LIN {X 0,Y 672.579,Z 201.622,A -85,B 0,C 180,E1 -3473.113,E2 -3473.113} C_VEL
LIN {X 0,Y 679.346,Z 218.804,A -85,B 0,C 180,E1 -3474.693,E2 -3474.693} C_VEL
LIN {X 0,Y 682.037,Z 226.59,A -85,B 0,C 180,E1 -3475.434,E2 -3475.434} C_VEL
LIN {X 0,Y 680.752,Z 266.781,A -85,B 0,C 180,E1 -3478.375,E2 -3478.375} C_VEL
LIN {X 0,Y 679.52,Z 306.415,A -85,B 0,C 180,E1 -3481.238,E2 -3481.238} C_VEL
LIN {X 0,Y 679.485,Z 310.379,A -85,B 0,C 180,E1 -3481.504,E2 -3481.504} C_VEL
LIN {X 0,Y 681.228,Z 320.364,A -85,B 0,C 180,E1 -3481.706,E2 -3481.706} C_VEL
LIN {X 0,Y 679.45,Z 568.033,A -85,B 0,C 180,E1 -3484.516,E2 -3484.516} C_VEL
LIN {X 0,Y 679.106,Z 608.658,A -85,B 0,C 180,E1 -3485,E2 -3485} C_VEL
LIN {X 0,Y 678.694,Z 631.405,A -85,B 0,C 180,E1 -3485.414,E2 -3485.414} C_VEL
LIN {X 0,Y 678.15,Z 652.378,A -85,B 0,C 180,E1 -3485.964,E2 -3485.964} C_VEL
LIN {X 0,Y 677.64,Z 669.474,A -85,B 0,C 180,E1 -3486.522,E2 -3486.522} C_VEL
LIN {X 0,Y 677.053,Z 686.549,A -85,B 0,C 180,E1 -3487.19,E2 -3487.19} C_VEL
LIN {X 0,Y 676.5,Z 702.61,A -85,B 0,C 180,E1 -3487.931,E2 -3487.931} C_VEL
LIN {X 0,Y 675.912,Z 718.028,A -85,B 0,C 180,E1 -3488.75,E2 -3488.75} C_VEL
LIN {X 0,Y 675.272,Z 734.049,A -85,B 0,C 180,E1 -3489.727,E2 -3489.727} C_VEL
LIN {X 0,Y 674.601,Z 751.677,A -85,B 0,C 180,E1 -3490.969,E2 -3490.969} C_VEL
LIN {X 0,Y 673.925,Z 768.647,A -85,B 0,C 180,E1 -3492.382,E2 -3492.382} C_VEL
LIN {X 0,Y 673.437,Z 781.527,A -85,B 0,C 180,E1 -3493.614,E2 -3493.614} C_VEL
LIN {X 0,Y 673.036,Z 793.645,A -85,B 0,C 180,E1 -3494.931,E2 -3494.931} C_VEL
LIN {X 0,Y 672.65,Z 806.255,A -85,B 0,C 180,E1 -3496.504,E2 -3496.504} C_VEL
LIN {X 0,Y 672.335,Z 818.497,A -85,B 0,C 180,E1 -3498.331,E2 -3498.331} C_VEL
LIN {X 0,Y 672.156,Z 827.245,A -85,B 0,C 180,E1 -3499.89,E2 -3499.89} C_VEL
LIN {X 0,Y 672.032,Z 834.911,A -85,B 0,C 180,E1 -3501.53,E2 -3501.53} C_VEL
LIN {X 0,Y 671.95,Z 841.394,A -85,B 0,C 180,E1 -3503.249,E2 -3503.249} C_VEL
LIN {X 0,Y 671.913,Z 846.943,A -85,B 0,C 180,E1 -3505.22,E2 -3505.22} C_VEL
LIN {X 0,Y 671.901,Z 850.246,A -85,B 0,C 180,E1 -3507.014,E2 -3507.014} C_VEL
LIN {X 0,Y 671.897,Z 851.95,A -85,B 0,C 180,E1 -3508.636,E2 -3508.636} C_VEL
LIN {X 0,Y 671.9,Z 852.431,A -85,B 0,C 180,E1 -3510.426,E2 -3510.426} C_VEL
LIN {X 0,Y 671.909,Z 851.064,A -85,B 0,C 180,E1 -3512.473,E2 -3512.473} C_VEL
LIN {X 0,Y 671.923,Z 848.206,A -85,B 0,C 180,E1 -3514.267,E2 -3514.267} C_VEL
LIN {X 0,Y 671.94,Z 844.025,A -85,B 0,C 180,E1 -3515.979,E2 -3515.979} C_VEL
LIN {X 0,Y 671.981,Z 838.375,A -85,B 0,C 180,E1 -3517.696,E2 -3517.696} C_VEL
LIN {X 0,Y 672.106,Z 829.893,A -85,B 0,C 180,E1 -3519.678,E2 -3519.678} C_VEL
LIN {X 0,Y 672.271,Z 821.072,A -85,B 0,C 180,E1 -3521.322,E2 -3521.322} C_VEL
LIN {X 0,Y 672.494,Z 811.756,A -85,B 0,C 180,E1 -3522.799,E2 -3522.799} C_VEL
LIN {X 0,Y 672.852,Z 799.566,A -85,B 0,C 180,E1 -3524.457,E2 -3524.457} C_VEL
LIN {X 0,Y 673.329,Z 784.965,A -85,B 0,C 180,E1 -3526.123,E2 -3526.123} C_VEL
LIN {X 0,Y 673.81,Z 771.549,A -85,B 0,C 180,E1 -3527.443,E2 -3527.443} C_VEL
LIN {X 0,Y 674.343,Z 757.55,A -85,B 0,C 180,E1 -3528.65,E2 -3528.65} C_VEL
LIN {X 0,Y 674.979,Z 741.859,A -85,B 0,C 180,E1 -3529.835,E2 -3529.835} C_VEL
LIN {X 0,Y 675.763,Z 721.934,A -85,B 0,C 180,E1 -3531.118,E2 -3531.118} C_VEL
LIN {X 0,Y 676.425,Z 704.738,A -85,B 0,C 180,E1 -3532.053,E2 -3532.053} C_VEL
LIN {X 0,Y 676.991,Z 688.587,A -85,B 0,C 180,E1 -3532.812,E2 -3532.812} C_VEL
LIN {X 0,Y 677.555,Z 671.856,A -85,B 0,C 180,E1 -3533.481,E2 -3533.481} C_VEL
LIN {X 0,Y 678.053,Z 655.221,A -85,B 0,C 180,E1 -3534.04,E2 -3534.04} C_VEL
LIN {X 0,Y 678.51,Z 638.285,A -85,B 0,C 180,E1 -3534.506,E2 -3534.506} C_VEL
LIN {X 0,Y 678.88,Z 621.075,A -85,B 0,C 180,E1 -3534.88,E2 -3534.88} C_VEL
LIN {X 0,Y 679.16,Z 603.568,A -85,B 0,C 180,E1 -3535.16,E2 -3535.16} C_VEL
LIN {X 0,Y 681.182,Z 326.681,A -85,B 0,C 180,E1 -3538.313,E2 -3538.313} C_VEL
LIN {X 0,Y 681.006,Z 317.975,A -85,B 0,C 180,E1 -3538.425,E2 -3538.425} C_VEL
LIN {X 0,Y 679.405,Z 309.493,A -85,B 0,C 180,E1 -3538.623,E2 -3538.623} C_VEL
LIN {X 0,Y 680.471,Z 276.701,A -85,B 0,C 180,E1 -3540.999,E2 -3540.999} C_VEL
LIN {X 0,Y 681.79,Z 234.937,A -85,B 0,C 180,E1 -3544.043,E2 -3544.043} C_VEL
LIN {X 0,Y 681.872,Z 225.908,A -85,B 0,C 180,E1 -3544.716,E2 -3544.716} C_VEL
LIN {X 0,Y 675.939,Z 210.334,A -85,B 0,C 180,E1 -3546.202,E2 -3546.202} C_VEL
LIN {X 0,Y 672.552,Z 201.457,A -85,B 0,C 180,E1 -3547.022,E2 -3547.022} C_VEL
LIN {X 0,Y 672.581,Z 201.453,A -85,B 0,C 180,E1 -3549.958,E2 -3549.958} C_VEL
LIN {X 0,Y 672.558,Z 201.452,A -85,B 0,C 180,E1 -3552.915,E2 -3552.915} C_VEL
LIN {X 0,Y 672.581,Z 201.448,A -85,B 0,C 180,E1 -3555.913,E2 -3555.913} C_VEL
LIN {X 0,Y 672.561,Z 201.45,A -85,B 0,C 180,E1 -3558.919,E2 -3558.919} C_VEL
LIN {X 0,Y 672.58,Z 201.45,A -85,B 0,C 180,E1 -3561.905,E2 -3561.905} C_VEL
LIN {X 0,Y 672.565,Z 201.448,A -85,B 0,C 180,E1 -3564.98,E2 -3564.98} C_VEL
LIN {X 0,Y 672.578,Z 201.451,A -85,B 0,C 180,E1 -3567.945,E2 -3567.945} C_VEL
LIN {X 0,Y 672.57,Z 201.443,A -85,B 0,C 180,E1 -3570.946,E2 -3570.946} C_VEL
LIN {X 0,Y 672.575,Z 201.452,A -85,B 0,C 180,E1 -3573.987,E2 -3573.987} C_VEL
LIN {X 0,Y 672.573,Z 201.435,A -85,B 0,C 180,E1 -3576.984,E2 -3576.984} C_VEL
LIN {X 0,Y 672.572,Z 201.448,A -85,B 0,C 180,E1 -3580.005,E2 -3580.005} C_VEL
LIN {X 0,Y 672.574,Z 201.438,A -85,B 0,C 180,E1 -3583.059,E2 -3583.059} C_VEL
LIN {X 0,Y 672.569,Z 201.445,A -85,B 0,C 180,E1 -3586.064,E2 -3586.064} C_VEL
LIN {X 0,Y 672.576,Z 201.439,A -85,B 0,C 180,E1 -3589.117,E2 -3589.117} C_VEL
LIN {X 0,Y 672.565,Z 201.446,A -85,B 0,C 180,E1 -3592.139,E2 -3592.139} C_VEL
LIN {X 0,Y 672.579,Z 201.437,A -85,B 0,C 180,E1 -3595.139,E2 -3595.139} C_VEL
LIN {X 0,Y 672.561,Z 201.448,A -85,B 0,C 180,E1 -3598.211,E2 -3598.211} C_VEL
LIN {X 0,Y 672.581,Z 201.432,A -85,B 0,C 180,E1 -3601.193,E2 -3601.193} C_VEL
LIN {X 0,Y 672.557,Z 201.451,A -85,B 0,C 180,E1 -3604.263,E2 -3604.263} C_VEL
LIN {X 0,Y 672.582,Z 201.433,A -85,B 0,C 180,E1 -3607.26,E2 -3607.26} C_VEL
LIN {X 0,Y 672.555,Z 201.452,A -85,B 0,C 180,E1 -3610.277,E2 -3610.277} C_VEL
LIN {X 0,Y 672.586,Z 201.445,A -85,B 0,C 180,E1 -3613.235,E2 -3613.235} C_VEL
LIN {X 0,Y 672.554,Z 201.454,A -85,B 0,C 180,E1 -3616.23,E2 -3616.23} C_VEL
LIN {X 0,Y 672.582,Z 201.444,A -85,B 0,C 180,E1 -3619.181,E2 -3619.181} C_VEL
LIN {X 0,Y 672.552,Z 201.454,A -85,B 0,C 180,E1 -3622.279,E2 -3622.279} C_VEL
LIN {X 0,Y 672.581,Z 201.446,A -85,B 0,C 180,E1 -3625.256,E2 -3625.256} C_VEL
LIN {X 0,Y 672.547,Z 201.453,A -85,B 0,C 180,E1 -3628.341,E2 -3628.341} C_VEL
LIN {X 0,Y 672.578,Z 201.447,A -85,B 0,C 180,E1 -3631.26,E2 -3631.26} C_VEL
LIN {X 0,Y 672.549,Z 201.455,A -85,B 0,C 180,E1 -3634.296,E2 -3634.296} C_VEL
LIN {X 0,Y 672.559,Z 201.449,A -85,B 0,C 180,E1 -3637.168,E2 -3637.168} C_VEL
LIN {X 0,Y 672.548,Z 201.456,A -85,B 0,C 180,E1 -3640.298,E2 -3640.298} C_VEL
LIN {X 0,Y 672.55,Z 201.452,A -85,B 0,C 180,E1 -3643.149,E2 -3643.149} C_VEL
LIN {X 0,Y 672.552,Z 201.458,A -85,B 0,C 180,E1 -3646.265,E2 -3646.265} C_VEL
LIN {X 0,Y 672.57,Z 201.682,A -85,B 0,C 180,E1 -3647.086,E2 -3647.086} C_VEL
LIN {X 0,Y 673.919,Z 205.007,A -85,B 0,C 180,E1 -3647.385,E2 -3647.385} C_VEL
LIN {X 0,Y 682.61,Z 222.727,A -85,B 0,C 180,E1 -3649.035,E2 -3649.035} C_VEL
LIN {X 0,Y 686.788,Z 232.051,A -85,B 0,C 180,E1 -3649.81,E2 -3649.81} C_VEL
LIN {X 0,Y 684.973,Z 290.804,A -85,B 0,C 180,E1 -3652.661,E2 -3652.661} C_VEL
LIN {X 0,Y 684.73,Z 300.754,A -85,B 0,C 180,E1 -3653.126,E2 -3653.126} C_VEL
LIN {X 0,Y 686.841,Z 315.173,A -85,B 0,C 180,E1 -3653.424,E2 -3653.424} C_VEL
LIN {X 0,Y 685.386,Z 510.12,A -85,B 0,C 180,E1 -3655.72,E2 -3655.72} C_VEL
LIN {X 0,Y 683.704,Z 691.141,A -85,B 0,C 180,E1 -3657.878,E2 -3657.878} C_VEL
LIN {X 0,Y 683.128,Z 716.495,A -85,B 0,C 180,E1 -3658.328,E2 -3658.328} C_VEL
LIN {X 0,Y 682.438,Z 738.1,A -85,B 0,C 180,E1 -3658.848,E2 -3658.848} C_VEL
LIN {X 0,Y 681.652,Z 761.266,A -85,B 0,C 180,E1 -3659.549,E2 -3659.549} C_VEL
LIN {X 0,Y 680.761,Z 782.216,A -85,B 0,C 180,E1 -3660.332,E2 -3660.332} C_VEL
LIN {X 0,Y 679.885,Z 802.279,A -85,B 0,C 180,E1 -3661.207,E2 -3661.207} C_VEL
LIN {X 0,Y 678.731,Z 825.506,A -85,B 0,C 180,E1 -3662.399,E2 -3662.399} C_VEL
LIN {X 0,Y 677.787,Z 844.732,A -85,B 0,C 180,E1 -3663.543,E2 -3663.543} C_VEL
LIN {X 0,Y 676.663,Z 866.009,A -85,B 0,C 180,E1 -3665,E2 -3665} C_VEL
LIN {X 0,Y 675.802,Z 883.401,A -85,B 0,C 180,E1 -3666.362,E2 -3666.362} C_VEL
LIN {X 0,Y 674.846,Z 902.606,A -85,B 0,C 180,E1 -3668.076,E2 -3668.076} C_VEL
LIN {X 0,Y 674.159,Z 917.749,A -85,B 0,C 180,E1 -3669.614,E2 -3669.614} C_VEL
LIN {X 0,Y 673.471,Z 933.816,A -85,B 0,C 180,E1 -3671.475,E2 -3671.475} C_VEL
LIN {X 0,Y 673.017,Z 946.526,A -85,B 0,C 180,E1 -3673.16,E2 -3673.16} C_VEL
LIN {X 0,Y 672.589,Z 959.764,A -85,B 0,C 180,E1 -3675.185,E2 -3675.185} C_VEL
LIN {X 0,Y 672.315,Z 969.606,A -85,B 0,C 180,E1 -3676.942,E2 -3676.942} C_VEL
LIN {X 0,Y 672.101,Z 979.477,A -85,B 0,C 180,E1 -3679.022,E2 -3679.022} C_VEL
LIN {X 0,Y 672.004,Z 986.514,A -85,B 0,C 180,E1 -3680.839,E2 -3680.839} C_VEL
LIN {X 0,Y 671.934,Z 992.507,A -85,B 0,C 180,E1 -3682.733,E2 -3682.733} C_VEL
LIN {X 0,Y 671.893,Z 997.337,A -85,B 0,C 180,E1 -3684.792,E2 -3684.792} C_VEL
LIN {X 0,Y 671.908,Z 1000.237,A -85,B 0,C 180,E1 -3686.587,E2 -3686.587} C_VEL
LIN {X 0,Y 671.908,Z 1002.17,A -85,B 0,C 180,E1 -3688.721,E2 -3688.721} C_VEL
LIN {X 0,Y 671.882,Z 1002.351,A -85,B 0,C 180,E1 -3690.597,E2 -3690.597} C_VEL
LIN {X 0,Y 671.907,Z 1001.363,A -85,B 0,C 180,E1 -3692.388,E2 -3692.388} C_VEL
LIN {X 0,Y 671.918,Z 998.608,A -85,B 0,C 180,E1 -3694.524,E2 -3694.524} C_VEL
LIN {X 0,Y 671.925,Z 994.689,A -85,B 0,C 180,E1 -3696.408,E2 -3696.408} C_VEL
LIN {X 0,Y 671.975,Z 989.201,A -85,B 0,C 180,E1 -3698.385,E2 -3698.385} C_VEL
LIN {X 0,Y 672.091,Z 981.605,A -85,B 0,C 180,E1 -3700.457,E2 -3700.457} C_VEL
LIN {X 0,Y 672.253,Z 973.118,A -85,B 0,C 180,E1 -3702.368,E2 -3702.368} C_VEL
LIN {X 0,Y 672.515,Z 962.354,A -85,B 0,C 180,E1 -3704.377,E2 -3704.377} C_VEL
LIN {X 0,Y 672.843,Z 951.388,A -85,B 0,C 180,E1 -3706.135,E2 -3706.135} C_VEL
LIN {X 0,Y 673.361,Z 936.945,A -85,B 0,C 180,E1 -3708.129,E2 -3708.129} C_VEL
LIN {X 0,Y 673.931,Z 922.728,A -85,B 0,C 180,E1 -3709.839,E2 -3709.839} C_VEL
LIN {X 0,Y 674.685,Z 906.31,A -85,B 0,C 180,E1 -3711.564,E2 -3711.564} C_VEL
LIN {X 0,Y 675.451,Z 890.139,A -85,B 0,C 180,E1 -3713.065,E2 -3713.065} C_VEL
LIN {X 0,Y 676.436,Z 870.867,A -85,B 0,C 180,E1 -3714.636,E2 -3714.636} C_VEL
LIN {X 0,Y 677.326,Z 853.071,A -85,B 0,C 180,E1 -3715.91,E2 -3715.91} C_VEL
LIN {X 0,Y 678.489,Z 830.879,A -85,B 0,C 180,E1 -3717.296,E2 -3717.296} C_VEL
LIN {X 0,Y 679.431,Z 811.337,A -85,B 0,C 180,E1 -3718.351,E2 -3718.351} C_VEL
LIN {X 0,Y 680.53,Z 787.863,A -85,B 0,C 180,E1 -3719.438,E2 -3719.438} C_VEL
LIN {X 0,Y 681.37,Z 767.685,A -85,B 0,C 180,E1 -3720.222,E2 -3720.222} C_VEL
LIN {X 0,Y 682.256,Z 745.15,A -85,B 0,C 180,E1 -3720.958,E2 -3720.958} C_VEL
LIN {X 0,Y 682.957,Z 721.163,A -85,B 0,C 180,E1 -3721.571,E2 -3721.571} C_VEL
LIN {X 0,Y 683.574,Z 698.388,A -85,B 0,C 180,E1 -3722.013,E2 -3722.013} C_VEL
LIN {X 0,Y 684.015,Z 664.777,A -85,B 0,C 180,E1 -3722.453,E2 -3722.453} C_VEL
LIN {X 0,Y 686.084,Z 426.859,A -85,B 0,C 180,E1 -3725.272,E2 -3725.272} C_VEL
LIN {X 0,Y 686.203,Z 312.509,A -85,B 0,C 180,E1 -3726.55,E2 -3726.55} C_VEL
LIN {X 0,Y 684.133,Z 300.68,A -85,B 0,C 180,E1 -3726.781,E2 -3726.781} C_VEL
LIN {X 0,Y 685,Z 265.459,A -85,B 0,C 180,E1 -3728.45,E2 -3728.45} C_VEL
LIN {X 0,Y 686.519,Z 233.708,A -85,B 0,C 180,E1 -3730.073,E2 -3730.073} C_VEL
LIN {X 0,Y 686.523,Z 231.357,A -85,B 0,C 180,E1 -3730.209,E2 -3730.209} C_VEL
LIN {X 0,Y 680.861,Z 218.547,A -85,B 0,C 180,E1 -3731.498,E2 -3731.498} C_VEL
LIN {X 0,Y 676.932,Z 210.351,A -85,B 0,C 180,E1 -3732.517,E2 -3732.517} C_VEL
LIN {X 0,Y 674.606,Z 205.849,A -85,B 0,C 180,E1 -3733.177,E2 -3733.177} C_VEL
LIN {X 0,Y 672.75,Z 202.49,A -85,B 0,C 180,E1 -3733.753,E2 -3733.753} C_VEL
LIN {X 0,Y 672.552,Z 201.458,A -85,B 0,C 180,E1 -3733.906,E2 -3733.906} C_VEL
LIN {X 0,Y 672.565,Z 201.456,A -85,B 0,C 180,E1 -3737.086,E2 -3737.086} C_VEL
LIN {X 0,Y 672.538,Z 201.46,A -85,B 0,C 180,E1 -3739.927,E2 -3739.927} C_VEL
LIN {X 0,Y 672.614,Z 201.669,A -85,B 0,C 180,E1 -3742.367,E2 -3742.367} C_VEL
LIN {X 0,Y 674.124,Z 205.273,A -85,B 0,C 180,E1 -3742.938,E2 -3742.938} C_VEL
LIN {X 0,Y 675.014,Z 206.813,A -85,B 0,C 180,E1 -3743.191,E2 -3743.191} C_VEL
LIN {X 0,Y 678.723,Z 215.05,A -85,B 0,C 180,E1 -3744.311,E2 -3744.311} C_VEL
LIN {X 0,Y 683.33,Z 226.73,A -85,B 0,C 180,E1 -3745.617,E2 -3745.617} C_VEL
LIN {X 0,Y 683.402,Z 229.375,A -85,B 0,C 180,E1 -3745.817,E2 -3745.817} C_VEL
LIN {X 0,Y 680.701,Z 272.496,A -85,B 0,C 180,E1 -3748.588,E2 -3748.588} C_VEL
LIN {X 0,Y 678.57,Z 326.363,A -85,B 0,C 180,E1 -3751.866,E2 -3751.866} C_VEL
LIN {X 0,Y 677.146,Z 378.659,A -85,B 0,C 180,E1 -3754.926,E2 -3754.926} C_VEL
LIN {X 0,Y 675.934,Z 433.54,A -85,B 0,C 180,E1 -3758.049,E2 -3758.049} C_VEL
LIN {X 0,Y 675.545,Z 457.444,A -85,B 0,C 180,E1 -3759.368,E2 -3759.368} C_VEL
LIN {X 0,Y 678.294,Z 481.315,A -85,B 0,C 180,E1 -3759.835,E2 -3759.835} C_VEL
LIN {X 0,Y 676.325,Z 608.391,A -85,B 0,C 180,E1 -3761.464,E2 -3761.464} C_VEL
LIN {X 0,Y 675.634,Z 682.185,A -85,B 0,C 180,E1 -3762.378,E2 -3762.378} C_VEL
LIN {X 0,Y 675.344,Z 701.727,A -85,B 0,C 180,E1 -3762.778,E2 -3762.778} C_VEL
LIN {X 0,Y 675.02,Z 719.823,A -85,B 0,C 180,E1 -3763.3,E2 -3763.3} C_VEL
LIN {X 0,Y 674.636,Z 737.26,A -85,B 0,C 180,E1 -3763.954,E2 -3763.954} C_VEL
LIN {X 0,Y 674.245,Z 754.12,A -85,B 0,C 180,E1 -3764.749,E2 -3764.749} C_VEL
LIN {X 0,Y 673.837,Z 770.294,A -85,B 0,C 180,E1 -3765.69,E2 -3765.69} C_VEL
LIN {X 0,Y 673.428,Z 785.113,A -85,B 0,C 180,E1 -3766.738,E2 -3766.738} C_VEL
LIN {X 0,Y 673.048,Z 798.81,A -85,B 0,C 180,E1 -3767.909,E2 -3767.909} C_VEL
LIN {X 0,Y 672.736,Z 810.592,A -85,B 0,C 180,E1 -3769.119,E2 -3769.119} C_VEL
LIN {X 0,Y 672.473,Z 821.059,A -85,B 0,C 180,E1 -3770.414,E2 -3770.414} C_VEL
LIN {X 0,Y 672.265,Z 830.19,A -85,B 0,C 180,E1 -3771.791,E2 -3771.791} C_VEL
LIN {X 0,Y 672.124,Z 837.938,A -85,B 0,C 180,E1 -3773.251,E2 -3773.251} C_VEL
LIN {X 0,Y 672.045,Z 844.23,A -85,B 0,C 180,E1 -3774.793,E2 -3774.793} C_VEL
LIN {X 0,Y 671.982,Z 848.97,A -85,B 0,C 180,E1 -3776.417,E2 -3776.417} C_VEL
LIN {X 0,Y 671.955,Z 852.015,A -85,B 0,C 180,E1 -3778.124,E2 -3778.124} C_VEL
LIN {X 0,Y 671.948,Z 853.148,A -85,B 0,C 180,E1 -3779.744,E2 -3779.744} C_VEL
LIN {X 0,Y 671.945,Z 852.596,A -85,B 0,C 180,E1 -3781.364,E2 -3781.364} C_VEL
LIN {X 0,Y 671.96,Z 850.344,A -85,B 0,C 180,E1 -3782.985,E2 -3782.985} C_VEL
LIN {X 0,Y 671.989,Z 846.324,A -85,B 0,C 180,E1 -3784.609,E2 -3784.609} C_VEL
LIN {X 0,Y 672.056,Z 840.398,A -85,B 0,C 180,E1 -3786.235,E2 -3786.235} C_VEL
LIN {X 0,Y 672.168,Z 832.667,A -85,B 0,C 180,E1 -3787.813,E2 -3787.813} C_VEL
LIN {X 0,Y 672.345,Z 823.743,A -85,B 0,C 180,E1 -3789.243,E2 -3789.243} C_VEL
LIN {X 0,Y 672.591,Z 813.122,A -85,B 0,C 180,E1 -3790.623,E2 -3790.623} C_VEL
LIN {X 0,Y 672.898,Z 800.975,A -85,B 0,C 180,E1 -3791.92,E2 -3791.92} C_VEL
LIN {X 0,Y 673.268,Z 787.237,A -85,B 0,C 180,E1 -3793.134,E2 -3793.134} C_VEL
LIN {X 0,Y 673.678,Z 772.328,A -85,B 0,C 180,E1 -3794.224,E2 -3794.224} C_VEL
LIN {X 0,Y 674.102,Z 756.538,A -85,B 0,C 180,E1 -3795.177,E2 -3795.177} C_VEL
LIN {X 0,Y 674.498,Z 739.713,A -85,B 0,C 180,E1 -3796.006,E2 -3796.006} C_VEL
LIN {X 0,Y 674.919,Z 721.886,A -85,B 0,C 180,E1 -3796.703,E2 -3796.703} C_VEL
LIN {X 0,Y 675.274,Z 702.619,A -85,B 0,C 180,E1 -3797.276,E2 -3797.276} C_VEL
LIN {X 0,Y 675.562,Z 683.284,A -85,B 0,C 180,E1 -3797.68,E2 -3797.68} C_VEL
LIN {X 0,Y 675.824,Z 651.623,A -85,B 0,C 180,E1 -3798.079,E2 -3798.079} C_VEL
LIN {X 0,Y 676.454,Z 561.656,A -85,B 0,C 180,E1 -3799.105,E2 -3799.105} C_VEL
LIN {X 0,Y 675.607,Z 554.064,A -85,B 0,C 180,E1 -3799.223,E2 -3799.223} C_VEL
LIN {X 0,Y 669.963,Z 534.195,A -85,B 0,C 180,E1 -3799.649,E2 -3799.649} C_VEL
LIN {X 0,Y 669.337,Z 527.67,A -85,B 0,C 180,E1 -3799.75,E2 -3799.75} C_VEL
LIN {X 0,Y 669.559,Z 478.594,A -85,B 0,C 180,E1 -3800.344,E2 -3800.344} C_VEL
LIN {X 0,Y 667.897,Z 464.609,A -85,B 0,C 180,E1 -3800.598,E2 -3800.598} C_VEL
LIN {X 0,Y 669.123,Z 409.096,A -85,B 0,C 180,E1 -3803.749,E2 -3803.749} C_VEL
LIN {X 0,Y 670.415,Z 355.832,A -85,B 0,C 180,E1 -3806.819,E2 -3806.819} C_VEL
LIN {X 0,Y 671.812,Z 303.955,A -85,B 0,C 180,E1 -3809.858,E2 -3809.858} C_VEL
LIN {X 0,Y 673.338,Z 252.657,A -85,B 0,C 180,E1 -3812.922,E2 -3812.922} C_VEL
LIN {X 0,Y 674.106,Z 227.628,A -85,B 0,C 180,E1 -3814.441,E2 -3814.441} C_VEL
LIN {X 0,Y 664.614,Z 202.433,A -85,B 0,C 180,E1 -3816.595,E2 -3816.595} C_VEL
LIN {X 0,Y 664.637,Z 202.442,A -85,B 0,C 180,E1 -3819.634,E2 -3819.634} C_VEL
LIN {X 0,Y 664.598,Z 202.446,A -85,B 0,C 180,E1 -3822.506,E2 -3822.506} C_VEL
LIN {X 0,Y 664.644,Z 202.437,A -85,B 0,C 180,E1 -3825.61,E2 -3825.61} C_VEL
LIN {X 0,Y 664.607,Z 202.442,A -85,B 0,C 180,E1 -3828.664,E2 -3828.664} C_VEL
LIN {X 0,Y 664.64,Z 202.444,A -85,B 0,C 180,E1 -3831.61,E2 -3831.61} C_VEL
LIN {X 0,Y 664.587,Z 202.509,A -85,B 0,C 180,E1 -3832.662,E2 -3832.662} C_VEL
LIN {X 0,Y 667.131,Z 208.973,A -85,B 0,C 180,E1 -3833.236,E2 -3833.236} C_VEL
LIN {X 0,Y 673.998,Z 226.544,A -85,B 0,C 180,E1 -3834.902,E2 -3834.902} C_VEL
LIN {X 0,Y 675.119,Z 230.081,A -85,B 0,C 180,E1 -3835.235,E2 -3835.235} C_VEL
LIN {X 0,Y 673.763,Z 269.836,A -85,B 0,C 180,E1 -3838.158,E2 -3838.158} C_VEL
LIN {X 0,Y 672.675,Z 312.651,A -85,B 0,C 180,E1 -3841.205,E2 -3841.205} C_VEL
LIN {X 0,Y 674.226,Z 321.813,A -85,B 0,C 180,E1 -3841.392,E2 -3841.392} C_VEL
LIN {X 0,Y 672.018,Z 576.504,A -85,B 0,C 180,E1 -3844.347,E2 -3844.347} C_VEL
LIN {X 0,Y 671.7,Z 612.862,A -85,B 0,C 180,E1 -3844.79,E2 -3844.79} C_VEL
LIN {X 0,Y 671.233,Z 635.63,A -85,B 0,C 180,E1 -3845.243,E2 -3845.243} C_VEL
LIN {X 0,Y 670.779,Z 653.07,A -85,B 0,C 180,E1 -3845.706,E2 -3845.706} C_VEL
LIN {X 0,Y 670.25,Z 669.467,A -85,B 0,C 180,E1 -3846.247,E2 -3846.247} C_VEL
LIN {X 0,Y 669.63,Z 686.01,A -85,B 0,C 180,E1 -3846.899,E2 -3846.899} C_VEL
LIN {X 0,Y 669.013,Z 702.077,A -85,B 0,C 180,E1 -3847.643,E2 -3847.643} C_VEL
LIN {X 0,Y 668.387,Z 717.241,A -85,B 0,C 180,E1 -3848.453,E2 -3848.453} C_VEL
LIN {X 0,Y 667.726,Z 732.366,A -85,B 0,C 180,E1 -3849.376,E2 -3849.376} C_VEL
LIN {X 0,Y 667.085,Z 746.814,A -85,B 0,C 180,E1 -3850.382,E2 -3850.382} C_VEL
LIN {X 0,Y 666.436,Z 762.21,A -85,B 0,C 180,E1 -3851.602,E2 -3851.602} C_VEL
LIN {X 0,Y 665.739,Z 778.959,A -85,B 0,C 180,E1 -3853.15,E2 -3853.15} C_VEL
LIN {X 0,Y 665.22,Z 792.126,A -85,B 0,C 180,E1 -3854.571,E2 -3854.571} C_VEL
LIN {X 0,Y 664.825,Z 803.575,A -85,B 0,C 180,E1 -3855.987,E2 -3855.987} C_VEL
LIN {X 0,Y 664.513,Z 814.084,A -85,B 0,C 180,E1 -3857.486,E2 -3857.486} C_VEL
LIN {X 0,Y 664.233,Z 825.477,A -85,B 0,C 180,E1 -3859.417,E2 -3859.417} C_VEL
LIN {X 0,Y 664.065,Z 833.798,A -85,B 0,C 180,E1 -3861.165,E2 -3861.165} C_VEL
LIN {X 0,Y 663.983,Z 839.878,A -85,B 0,C 180,E1 -3862.733,E2 -3862.733} C_VEL
LIN {X 0,Y 663.933,Z 844.97,A -85,B 0,C 180,E1 -3864.382,E2 -3864.382} C_VEL
LIN {X 0,Y 663.918,Z 849.209,A -85,B 0,C 180,E1 -3866.287,E2 -3866.287} C_VEL
LIN {X 0,Y 663.913,Z 851.709,A -85,B 0,C 180,E1 -3868.274,E2 -3868.274} C_VEL
LIN {X 0,Y 663.919,Z 852.424,A -85,B 0,C 180,E1 -3870,E2 -3870} C_VEL
LIN {X 0,Y 663.911,Z 851.771,A -85,B 0,C 180,E1 -3871.726,E2 -3871.726} C_VEL
LIN {X 0,Y 663.917,Z 849.529,A -85,B 0,C 180,E1 -3873.627,E2 -3873.627} C_VEL
LIN {X 0,Y 663.936,Z 845.22,A -85,B 0,C 180,E1 -3875.618,E2 -3875.618} C_VEL
LIN {X 0,Y 663.98,Z 840.192,A -85,B 0,C 180,E1 -3877.267,E2 -3877.267} C_VEL
LIN {X 0,Y 664.054,Z 834.18,A -85,B 0,C 180,E1 -3878.835,E2 -3878.835} C_VEL
LIN {X 0,Y 664.223,Z 825.939,A -85,B 0,C 180,E1 -3880.583,E2 -3880.583} C_VEL
LIN {X 0,Y 664.494,Z 814.683,A -85,B 0,C 180,E1 -3882.514,E2 -3882.514} C_VEL
LIN {X 0,Y 664.807,Z 804.016,A -85,B 0,C 180,E1 -3884.045,E2 -3884.045} C_VEL
LIN {X 0,Y 665.191,Z 792.891,A -85,B 0,C 180,E1 -3885.43,E2 -3885.43} C_VEL
LIN {X 0,Y 665.655,Z 780.673,A -85,B 0,C 180,E1 -3886.763,E2 -3886.763} C_VEL
LIN {X 0,Y 666.33,Z 764.724,A -85,B 0,C 180,E1 -3888.278,E2 -3888.278} C_VEL
LIN {X 0,Y 667.041,Z 748.021,A -85,B 0,C 180,E1 -3889.62,E2 -3889.62} C_VEL
LIN {X 0,Y 667.68,Z 733.331,A -85,B 0,C 180,E1 -3890.651,E2 -3890.651} C_VEL
LIN {X 0,Y 668.355,Z 717.99,A -85,B 0,C 180,E1 -3891.594,E2 -3891.594} C_VEL
LIN {X 0,Y 668.982,Z 702.926,A -85,B 0,C 180,E1 -3892.404,E2 -3892.404} C_VEL
LIN {X 0,Y 669.569,Z 687.517,A -85,B 0,C 180,E1 -3893.125,E2 -3893.125} C_VEL
LIN {X 0,Y 670.158,Z 671.819,A -85,B 0,C 180,E1 -3893.756,E2 -3893.756} C_VEL
LIN {X 0,Y 670.68,Z 655.903,A -85,B 0,C 180,E1 -3894.298,E2 -3894.298} C_VEL
LIN {X 0,Y 671.137,Z 639.382,A -85,B 0,C 180,E1 -3894.755,E2 -3894.755} C_VEL
LIN {X 0,Y 671.516,Z 621.739,A -85,B 0,C 180,E1 -3895.139,E2 -3895.139} C_VEL
LIN {X 0,Y 671.791,Z 603.592,A -85,B 0,C 180,E1 -3895.427,E2 -3895.427} C_VEL
LIN {X 0,Y 673.859,Z 361.059,A -85,B 0,C 180,E1 -3898.242,E2 -3898.242} C_VEL
LIN {X 0,Y 674.06,Z 319.616,A -85,B 0,C 180,E1 -3898.735,E2 -3898.735} C_VEL
LIN {X 0,Y 672.599,Z 311.902,A -85,B 0,C 180,E1 -3898.915,E2 -3898.915} C_VEL
LIN {X 0,Y 673.656,Z 272.529,A -85,B 0,C 180,E1 -3901.735,E2 -3901.735} C_VEL
LIN {X 0,Y 675.029,Z 233.352,A -85,B 0,C 180,E1 -3904.615,E2 -3904.615} C_VEL
LIN {X 0,Y 674.99,Z 229.369,A -85,B 0,C 180,E1 -3904.915,E2 -3904.915} C_VEL
LIN {X 0,Y 668.438,Z 212.229,A -85,B 0,C 180,E1 -3906.555,E2 -3906.555} C_VEL
LIN {X 0,Y 664.641,Z 202.534,A -85,B 0,C 180,E1 -3907.429,E2 -3907.429} C_VEL
LIN {X 0,Y 664.632,Z 202.437,A -85,B 0,C 180,E1 -3910.648,E2 -3910.648} C_VEL
LIN {X 0,Y 664.643,Z 202.438,A -85,B 0,C 180,E1 -3913.671,E2 -3913.671} C_VEL
LIN {X 0,Y 664.627,Z 202.434,A -85,B 0,C 180,E1 -3916.802,E2 -3916.802} C_VEL
LIN {X 0,Y 664.645,Z 202.437,A -85,B 0,C 180,E1 -3919.839,E2 -3919.839} C_VEL
LIN {X 0,Y 664.628,Z 202.433,A -85,B 0,C 180,E1 -3922.895,E2 -3922.895} C_VEL
LIN {X 0,Y 664.637,Z 202.436,A -85,B 0,C 180,E1 -3925.969,E2 -3925.969} C_VEL
LIN {X 0,Y 664.626,Z 202.437,A -85,B 0,C 180,E1 -3929.04,E2 -3929.04} C_VEL
LIN {X 0,Y 664.636,Z 202.435,A -85,B 0,C 180,E1 -3932.018,E2 -3932.018} C_VEL
LIN {X 0,Y 664.629,Z 202.436,A -85,B 0,C 180,E1 -3935.087,E2 -3935.087} C_VEL
LIN {X 0,Y 664.633,Z 202.439,A -85,B 0,C 180,E1 -3938.093,E2 -3938.093} C_VEL
LIN {X 0,Y 664.632,Z 202.431,A -85,B 0,C 180,E1 -3941.135,E2 -3941.135} C_VEL
LIN {X 0,Y 664.63,Z 202.44,A -85,B 0,C 180,E1 -3944.109,E2 -3944.109} C_VEL
LIN {X 0,Y 664.635,Z 202.428,A -85,B 0,C 180,E1 -3947.135,E2 -3947.135} C_VEL
LIN {X 0,Y 664.625,Z 202.44,A -85,B 0,C 180,E1 -3950.212,E2 -3950.212} C_VEL
LIN {X 0,Y 664.636,Z 202.431,A -85,B 0,C 180,E1 -3953.261,E2 -3953.261} C_VEL
LIN {X 0,Y 664.621,Z 202.439,A -85,B 0,C 180,E1 -3956.291,E2 -3956.291} C_VEL
LIN {X 0,Y 664.637,Z 202.434,A -85,B 0,C 180,E1 -3959.31,E2 -3959.31} C_VEL
LIN {X 0,Y 664.616,Z 202.438,A -85,B 0,C 180,E1 -3962.328,E2 -3962.328} C_VEL
LIN {X 0,Y 664.641,Z 202.436,A -85,B 0,C 180,E1 -3965.352,E2 -3965.352} C_VEL
LIN {X 0,Y 664.615,Z 202.437,A -85,B 0,C 180,E1 -3968.304,E2 -3968.304} C_VEL
LIN {X 0,Y 664.645,Z 202.435,A -85,B 0,C 180,E1 -3971.278,E2 -3971.278} C_VEL
LIN {X 0,Y 664.613,Z 202.439,A -85,B 0,C 180,E1 -3974.332,E2 -3974.332} C_VEL
LIN {X 0,Y 664.647,Z 202.436,A -85,B 0,C 180,E1 -3977.33,E2 -3977.33} C_VEL
LIN {X 0,Y 664.608,Z 202.44,A -85,B 0,C 180,E1 -3980.398,E2 -3980.398} C_VEL
LIN {X 0,Y 664.649,Z 202.437,A -85,B 0,C 180,E1 -3983.411,E2 -3983.411} C_VEL
LIN {X 0,Y 664.604,Z 202.438,A -85,B 0,C 180,E1 -3986.47,E2 -3986.47} C_VEL
LIN {X 0,Y 664.65,Z 202.436,A -85,B 0,C 180,E1 -3989.468,E2 -3989.468} C_VEL
LIN {X 0,Y 664.601,Z 202.443,A -85,B 0,C 180,E1 -3992.487,E2 -3992.487} C_VEL
LIN {X 0,Y 664.643,Z 202.438,A -85,B 0,C 180,E1 -3995.394,E2 -3995.394} C_VEL
LIN {X 0,Y 664.601,Z 202.444,A -85,B 0,C 180,E1 -3998.416,E2 -3998.416} C_VEL
LIN {X 0,Y 664.633,Z 202.439,A -85,B 0,C 180,E1 -4001.334,E2 -4001.334} C_VEL
LIN {X 0,Y 664.601,Z 202.446,A -85,B 0,C 180,E1 -4004.394,E2 -4004.394} C_VEL
LIN {X 0,Y 664.612,Z 202.564,A -85,B 0,C 180,E1 -4006.495,E2 -4006.495} C_VEL
LIN {X 0,Y 665.771,Z 205.742,A -85,B 0,C 180,E1 -4006.777,E2 -4006.777} C_VEL
LIN {X 0,Y 667.227,Z 208.56,A -85,B 0,C 180,E1 -4007.059,E2 -4007.059} C_VEL
LIN {X 0,Y 673.156,Z 220.579,A -85,B 0,C 180,E1 -4008.216,E2 -4008.216} C_VEL
LIN {X 0,Y 679.957,Z 234.951,A -85,B 0,C 180,E1 -4009.487,E2 -4009.487} C_VEL
LIN {X 0,Y 680.142,Z 237.631,A -85,B 0,C 180,E1 -4009.64,E2 -4009.64} C_VEL
LIN {X 0,Y 678.085,Z 294.371,A -85,B 0,C 180,E1 -4012.429,E2 -4012.429} C_VEL
LIN {X 0,Y 677.934,Z 301.386,A -85,B 0,C 180,E1 -4012.754,E2 -4012.754} C_VEL
LIN {X 0,Y 680.085,Z 316.368,A -85,B 0,C 180,E1 -4013.074,E2 -4013.074} C_VEL
LIN {X 0,Y 678.07,Z 580.867,A -85,B 0,C 180,E1 -4016.186,E2 -4016.186} C_VEL
LIN {X 0,Y 676.916,Z 691.712,A -85,B 0,C 180,E1 -4017.525,E2 -4017.525} C_VEL
LIN {X 0,Y 676.278,Z 717.014,A -85,B 0,C 180,E1 -4017.982,E2 -4017.982} C_VEL
LIN {X 0,Y 675.543,Z 738.337,A -85,B 0,C 180,E1 -4018.501,E2 -4018.501} C_VEL
LIN {X 0,Y 674.614,Z 762.547,A -85,B 0,C 180,E1 -4019.246,E2 -4019.246} C_VEL
LIN {X 0,Y 673.652,Z 783.343,A -85,B 0,C 180,E1 -4020.036,E2 -4020.036} C_VEL
LIN {X 0,Y 672.656,Z 804.171,A -85,B 0,C 180,E1 -4020.961,E2 -4020.961} C_VEL
LIN {X 0,Y 671.429,Z 826.314,A -85,B 0,C 180,E1 -4022.121,E2 -4022.121} C_VEL
LIN {X 0,Y 670.361,Z 846.189,A -85,B 0,C 180,E1 -4023.323,E2 -4023.323} C_VEL
LIN {X 0,Y 669.167,Z 866.614,A -85,B 0,C 180,E1 -4024.748,E2 -4024.748} C_VEL
LIN {X 0,Y 668.23,Z 883.681,A -85,B 0,C 180,E1 -4026.101,E2 -4026.101} C_VEL
LIN {X 0,Y 667.192,Z 902.606,A -85,B 0,C 180,E1 -4027.811,E2 -4027.811} C_VEL
LIN {X 0,Y 666.423,Z 917.633,A -85,B 0,C 180,E1 -4029.354,E2 -4029.354} C_VEL
LIN {X 0,Y 665.657,Z 933.818,A -85,B 0,C 180,E1 -4031.249,E2 -4031.249} C_VEL
LIN {X 0,Y 665.151,Z 946.527,A -85,B 0,C 180,E1 -4032.955,E2 -4032.955} C_VEL
LIN {X 0,Y 664.668,Z 959.765,A -85,B 0,C 180,E1 -4035.004,E2 -4035.004} C_VEL
LIN {X 0,Y 664.363,Z 969.565,A -85,B 0,C 180,E1 -4036.776,E2 -4036.776} C_VEL
LIN {X 0,Y 664.133,Z 979.122,A -85,B 0,C 180,E1 -4038.801,E2 -4038.801} C_VEL
LIN {X 0,Y 664.025,Z 986.514,A -85,B 0,C 180,E1 -4040.728,E2 -4040.728} C_VEL
LIN {X 0,Y 663.938,Z 992.761,A -85,B 0,C 180,E1 -4042.732,E2 -4042.732} C_VEL
LIN {X 0,Y 663.894,Z 997.496,A -85,B 0,C 180,E1 -4044.815,E2 -4044.815} C_VEL
LIN {X 0,Y 663.905,Z 1000.35,A -85,B 0,C 180,E1 -4046.633,E2 -4046.633} C_VEL
LIN {X 0,Y 663.911,Z 1002.193,A -85,B 0,C 180,E1 -4048.792,E2 -4048.792} C_VEL
LIN {X 0,Y 663.884,Z 1002.328,A -85,B 0,C 180,E1 -4050.69,E2 -4050.69} C_VEL
LIN {X 0,Y 663.891,Z 1001.226,A -85,B 0,C 180,E1 -4052.59,E2 -4052.59} C_VEL
LIN {X 0,Y 663.91,Z 998.291,A -85,B 0,C 180,E1 -4054.752,E2 -4054.752} C_VEL
LIN {X 0,Y 663.93,Z 994.483,A -85,B 0,C 180,E1 -4056.572,E2 -4056.572} C_VEL
LIN {X 0,Y 663.978,Z 988.634,A -85,B 0,C 180,E1 -4058.661,E2 -4058.661} C_VEL
LIN {X 0,Y 664.107,Z 981.604,A -85,B 0,C 180,E1 -4060.585,E2 -4060.585} C_VEL
LIN {X 0,Y 664.295,Z 973.119,A -85,B 0,C 180,E1 -4062.518,E2 -4062.518} C_VEL
LIN {X 0,Y 664.592,Z 962.352,A -85,B 0,C 180,E1 -4064.552,E2 -4064.552} C_VEL
LIN {X 0,Y 664.955,Z 951.39,A -85,B 0,C 180,E1 -4066.331,E2 -4066.331} C_VEL
LIN {X 0,Y 665.521,Z 937.327,A -85,B 0,C 180,E1 -4068.301,E2 -4068.301} C_VEL
LIN {X 0,Y 666.104,Z 924.081,A -85,B 0,C 180,E1 -4069.923,E2 -4069.923} C_VEL
LIN {X 0,Y 667.003,Z 906.308,A -85,B 0,C 180,E1 -4071.825,E2 -4071.825} C_VEL
LIN {X 0,Y 667.853,Z 890.292,A -85,B 0,C 180,E1 -4073.329,E2 -4073.329} C_VEL
LIN {X 0,Y 668.965,Z 870.26,A -85,B 0,C 180,E1 -4074.977,E2 -4074.977} C_VEL
LIN {X 0,Y 670.028,Z 851.732,A -85,B 0,C 180,E1 -4076.309,E2 -4076.309} C_VEL
LIN {X 0,Y 671.229,Z 830.362,A -85,B 0,C 180,E1 -4077.647,E2 -4077.647} C_VEL
LIN {X 0,Y 672.271,Z 810.751,A -85,B 0,C 180,E1 -4078.712,E2 -4078.712} C_VEL
LIN {X 0,Y 673.505,Z 786.733,A -85,B 0,C 180,E1 -4079.825,E2 -4079.825} C_VEL
LIN {X 0,Y 674.376,Z 767.681,A -85,B 0,C 180,E1 -4080.568,E2 -4080.568} C_VEL
LIN {X 0,Y 675.344,Z 744.914,A -85,B 0,C 180,E1 -4081.319,E2 -4081.319} C_VEL
LIN {X 0,Y 676.124,Z 721.009,A -85,B 0,C 180,E1 -4081.931,E2 -4081.931} C_VEL
LIN {X 0,Y 676.788,Z 698.224,A -85,B 0,C 180,E1 -4082.376,E2 -4082.376} C_VEL
LIN {X 0,Y 677.267,Z 664.299,A -85,B 0,C 180,E1 -4082.823,E2 -4082.823} C_VEL
LIN {X 0,Y 678.641,Z 503.836,A -85,B 0,C 180,E1 -4084.713,E2 -4084.713} C_VEL
LIN {X 0,Y 679.056,Z 314.132,A -85,B 0,C 180,E1 -4086.821,E2 -4086.821} C_VEL
LIN {X 0,Y 677.02,Z 302.362,A -85,B 0,C 180,E1 -4087.055,E2 -4087.055} C_VEL
LIN {X 0,Y 678.296,Z 263.394,A -85,B 0,C 180,E1 -4088.955,E2 -4088.955} C_VEL
LIN {X 0,Y 680.073,Z 235.309,A -85,B 0,C 180,E1 -4090.459,E2 -4090.459} C_VEL
LIN {X 0,Y 674.941,Z 223.486,A -85,B 0,C 180,E1 -4091.699,E2 -4091.699} C_VEL
LIN {X 0,Y 671.142,Z 215.513,A -85,B 0,C 180,E1 -4092.736,E2 -4092.736} C_VEL
LIN {X 0,Y 669.286,Z 211.675,A -85,B 0,C 180,E1 -4093.317,E2 -4093.317} C_VEL
LIN {X 0,Y 667.505,Z 208.267,A -85,B 0,C 180,E1 -4093.912,E2 -4093.912} C_VEL
LIN {X 0,Y 666.66,Z 206.857,A -85,B 0,C 180,E1 -4094.198,E2 -4094.198} C_VEL
LIN {X 0,Y 664.748,Z 203.215,A -85,B 0,C 180,E1 -4095.012,E2 -4095.012} C_VEL
LIN {X 0,Y 664.604,Z 202.447,A -85,B 0,C 180,E1 -4095.176,E2 -4095.176} C_VEL
LIN {X 0,Y 664.63,Z 202.445,A -85,B 0,C 180,E1 -4098.089,E2 -4098.089} C_VEL
LIN {X 0,Y 664.619,Z 202.542,A -85,B 0,C 180,E1 -4101.144,E2 -4101.144} C_VEL
LIN {X 0,Y 666.113,Z 206.162,A -85,B 0,C 180,E1 -4101.906,E2 -4101.906} C_VEL
LIN {X 0,Y 667.299,Z 207.884,A -85,B 0,C 180,E1 -4102.294,E2 -4102.294} C_VEL
LIN {X 0,Y 669.667,Z 213.106,A -85,B 0,C 180,E1 -4103.16,E2 -4103.16} C_VEL
LIN {X 0,Y 672.856,Z 220.2,A -85,B 0,C 180,E1 -4104.161,E2 -4104.161} C_VEL
LIN {X 0,Y 677.01,Z 231.189,A -85,B 0,C 180,E1 -4105.432,E2 -4105.432} C_VEL
LIN {X 0,Y 673.983,Z 271.912,A -85,B 0,C 180,E1 -4108.12,E2 -4108.12} C_VEL
LIN {X 0,Y 671.543,Z 323.07,A -85,B 0,C 180,E1 -4111.302,E2 -4111.302} C_VEL
LIN {X 0,Y 669.914,Z 373.381,A -85,B 0,C 180,E1 -4114.304,E2 -4114.304} C_VEL
LIN {X 0,Y 668.512,Z 427.545,A -85,B 0,C 180,E1 -4117.44,E2 -4117.44} C_VEL
LIN {X 0,Y 668.026,Z 454.865,A -85,B 0,C 180,E1 -4118.969,E2 -4118.969} C_VEL
LIN {X 0,Y 671.143,Z 482.14,A -85,B 0,C 180,E1 -4119.537,E2 -4119.537} C_VEL
LIN {X 0,Y 668.827,Z 611.23,A -85,B 0,C 180,E1 -4121.252,E2 -4121.252} C_VEL
LIN {X 0,Y 668.046,Z 682.529,A -85,B 0,C 180,E1 -4122.164,E2 -4122.164} C_VEL
LIN {X 0,Y 667.722,Z 702.22,A -85,B 0,C 180,E1 -4122.576,E2 -4122.576} C_VEL
LIN {X 0,Y 667.369,Z 720.269,A -85,B 0,C 180,E1 -4123.102,E2 -4123.102} C_VEL
LIN {X 0,Y 666.928,Z 738.747,A -85,B 0,C 180,E1 -4123.808,E2 -4123.808} C_VEL
LIN {X 0,Y 666.499,Z 756.092,A -85,B 0,C 180,E1 -4124.646,E2 -4124.646} C_VEL
LIN {X 0,Y 666.055,Z 772.357,A -85,B 0,C 180,E1 -4125.614,E2 -4125.614} C_VEL
LIN {X 0,Y 665.628,Z 786.962,A -85,B 0,C 180,E1 -4126.668,E2 -4126.668} C_VEL
LIN {X 0,Y 665.228,Z 800.57,A -85,B 0,C 180,E1 -4127.852,E2 -4127.852} C_VEL
LIN {X 0,Y 664.886,Z 812.622,A -85,B 0,C 180,E1 -4129.118,E2 -4129.118} C_VEL
LIN {X 0,Y 664.596,Z 823.273,A -85,B 0,C 180,E1 -4130.474,E2 -4130.474} C_VEL
LIN {X 0,Y 664.372,Z 832.203,A -85,B 0,C 180,E1 -4131.867,E2 -4131.867} C_VEL
LIN {X 0,Y 664.22,Z 839.764,A -85,B 0,C 180,E1 -4133.344,E2 -4133.344} C_VEL
LIN {X 0,Y 664.134,Z 845.878,A -85,B 0,C 180,E1 -4134.904,E2 -4134.904} C_VEL
LIN {X 0,Y 664.059,Z 850.44,A -85,B 0,C 180,E1 -4136.547,E2 -4136.547} C_VEL
LIN {X 0,Y 664.028,Z 853.189,A -85,B 0,C 180,E1 -4138.188,E2 -4138.188} C_VEL
LIN {X 0,Y 664.017,Z 854.212,A -85,B 0,C 180,E1 -4139.827,E2 -4139.827} C_VEL
LIN {X 0,Y 664.009,Z 853.537,A -85,B 0,C 180,E1 -4141.467,E2 -4141.467} C_VEL
LIN {X 0,Y 664.027,Z 851.145,A -85,B 0,C 180,E1 -4143.107,E2 -4143.107} C_VEL
LIN {X 0,Y 664.059,Z 846.969,A -85,B 0,C 180,E1 -4144.75,E2 -4144.75} C_VEL
LIN {X 0,Y 664.132,Z 841.242,A -85,B 0,C 180,E1 -4146.31,E2 -4146.31} C_VEL
LIN {X 0,Y 664.255,Z 833.626,A -85,B 0,C 180,E1 -4147.873,E2 -4147.873} C_VEL
LIN {X 0,Y 664.456,Z 824.453,A -85,B 0,C 180,E1 -4149.353,E2 -4149.353} C_VEL
LIN {X 0,Y 664.725,Z 813.761,A -85,B 0,C 180,E1 -4150.75,E2 -4150.75} C_VEL
LIN {X 0,Y 665.06,Z 801.543,A -85,B 0,C 180,E1 -4152.063,E2 -4152.063} C_VEL
LIN {X 0,Y 665.464,Z 787.735,A -85,B 0,C 180,E1 -4153.291,E2 -4153.291} C_VEL
LIN {X 0,Y 665.907,Z 772.827,A -85,B 0,C 180,E1 -4154.389,E2 -4154.389} C_VEL
LIN {X 0,Y 666.365,Z 756.903,A -85,B 0,C 180,E1 -4155.358,E2 -4155.358} C_VEL
LIN {X 0,Y 666.799,Z 740.025,A -85,B 0,C 180,E1 -4156.195,E2 -4156.195} C_VEL
LIN {X 0,Y 667.255,Z 722.177,A -85,B 0,C 180,E1 -4156.901,E2 -4156.901} C_VEL
LIN {X 0,Y 667.644,Z 702.845,A -85,B 0,C 180,E1 -4157.482,E2 -4157.482} C_VEL
LIN {X 0,Y 667.965,Z 683.249,A -85,B 0,C 180,E1 -4157.896,E2 -4157.896} C_VEL
LIN {X 0,Y 668.246,Z 651.707,A -85,B 0,C 180,E1 -4158.298,E2 -4158.298} C_VEL
LIN {X 0,Y 669.337,Z 527.67,A -85,B 0,C 180,E1 -4159.75,E2 -4159.75} C_VEL
LIN {X 0,Y 668.499,Z 520.085,A -85,B 0,C 180,E1 -4159.873,E2 -4159.873} C_VEL
LIN {X 0,Y 662.906,Z 500.254,A -85,B 0,C 180,E1 -4160.321,E2 -4160.321} C_VEL
LIN {X 0,Y 662.276,Z 493.734,A -85,B 0,C 180,E1 -4160.426,E2 -4160.426} C_VEL
LIN {X 0,Y 662.163,Z 479.253,A -85,B 0,C 180,E1 -4160.611,E2 -4160.611} C_VEL
LIN {X 0,Y 660.317,Z 463.951,A -85,B 0,C 180,E1 -4160.885,E2 -4160.885} C_VEL
LIN {X 0,Y 661.651,Z 408.238,A -85,B 0,C 180,E1 -4164.081,E2 -4164.081} C_VEL
LIN {X 0,Y 663.089,Z 354.866,A -85,B 0,C 180,E1 -4167.188,E2 -4167.188} C_VEL
LIN {X 0,Y 664.656,Z 302.168,A -85,B 0,C 180,E1 -4170.313,E2 -4170.313} C_VEL
LIN {X 0,Y 666.284,Z 251.53,A -85,B 0,C 180,E1 -4173.368,E2 -4173.368} C_VEL
LIN {X 0,Y 666.861,Z 230.371,A -85,B 0,C 180,E1 -4174.672,E2 -4174.672} C_VEL
LIN {X 0,Y 657.644,Z 206.367,A -85,B 0,C 180,E1 -4176.749,E2 -4176.749} C_VEL
LIN {X 0,Y 656.679,Z 203.425,A -85,B 0,C 180,E1 -4177.028,E2 -4177.028} C_VEL
LIN {X 0,Y 656.639,Z 203.437,A -85,B 0,C 180,E1 -4180.214,E2 -4180.214} C_VEL
LIN {X 0,Y 656.707,Z 203.429,A -85,B 0,C 180,E1 -4183.043,E2 -4183.043} C_VEL
LIN {X 0,Y 656.698,Z 203.431,A -85,B 0,C 180,E1 -4186.149,E2 -4186.149} C_VEL
LIN {X 0,Y 656.67,Z 203.429,A -85,B 0,C 180,E1 -4189.099,E2 -4189.099} C_VEL
LIN {X 0,Y 656.659,Z 203.571,A -85,B 0,C 180,E1 -4192.212,E2 -4192.212} C_VEL
LIN {X 0,Y 659.411,Z 210.425,A -85,B 0,C 180,E1 -4192.829,E2 -4192.829} C_VEL
LIN {X 0,Y 666.925,Z 229.465,A -85,B 0,C 180,E1 -4194.647,E2 -4194.647} C_VEL
LIN {X 0,Y 668.197,Z 233.521,A -85,B 0,C 180,E1 -4195.032,E2 -4195.032} C_VEL
LIN {X 0,Y 666.824,Z 271.489,A -85,B 0,C 180,E1 -4197.838,E2 -4197.838} C_VEL
LIN {X 0,Y 665.888,Z 314.948,A -85,B 0,C 180,E1 -4200.9,E2 -4200.9} C_VEL
LIN {X 0,Y 667.246,Z 323.21,A -85,B 0,C 180,E1 -4201.069,E2 -4201.069} C_VEL
LIN {X 0,Y 664.264,Z 610.518,A -85,B 0,C 180,E1 -4204.508,E2 -4204.508} C_VEL
LIN {X 0,Y 663.816,Z 633.766,A -85,B 0,C 180,E1 -4204.944,E2 -4204.944} C_VEL
LIN {X 0,Y 663.244,Z 654.864,A -85,B 0,C 180,E1 -4205.507,E2 -4205.507} C_VEL
LIN {X 0,Y 662.667,Z 672.683,A -85,B 0,C 180,E1 -4206.105,E2 -4206.105} C_VEL
LIN {X 0,Y 661.959,Z 691.537,A -85,B 0,C 180,E1 -4206.875,E2 -4206.875} C_VEL
LIN {X 0,Y 661.069,Z 712.535,A -85,B 0,C 180,E1 -4207.922,E2 -4207.922} C_VEL
LIN {X 0,Y 660.244,Z 729.899,A -85,B 0,C 180,E1 -4208.966,E2 -4208.966} C_VEL
LIN {X 0,Y 659.542,Z 744.37,A -85,B 0,C 180,E1 -4209.963,E2 -4209.963} C_VEL
LIN {X 0,Y 658.871,Z 758.265,A -85,B 0,C 180,E1 -4211.049,E2 -4211.049} C_VEL
LIN {X 0,Y 658.262,Z 771.53,A -85,B 0,C 180,E1 -4212.223,E2 -4212.223} C_VEL
LIN {X 0,Y 657.696,Z 784.093,A -85,B 0,C 180,E1 -4213.483,E2 -4213.483} C_VEL
LIN {X 0,Y 657.144,Z 798.156,A -85,B 0,C 180,E1 -4215.099,E2 -4215.099} C_VEL
LIN {X 0,Y 656.69,Z 810.559,A -85,B 0,C 180,E1 -4216.797,E2 -4216.797} C_VEL
LIN {X 0,Y 656.397,Z 820.029,A -85,B 0,C 180,E1 -4218.311,E2 -4218.311} C_VEL
LIN {X 0,Y 656.196,Z 828.283,A -85,B 0,C 180,E1 -4219.853,E2 -4219.853} C_VEL
LIN {X 0,Y 656.053,Z 835.862,A -85,B 0,C 180,E1 -4221.551,E2 -4221.551} C_VEL
LIN {X 0,Y 655.959,Z 843.283,A -85,B 0,C 180,E1 -4223.699,E2 -4223.699} C_VEL
LIN {X 0,Y 655.92,Z 847.65,A -85,B 0,C 180,E1 -4225.453,E2 -4225.453} C_VEL
LIN {X 0,Y 655.905,Z 850.476,A -85,B 0,C 180,E1 -4227.116,E2 -4227.116} C_VEL
LIN {X 0,Y 655.898,Z 852.06,A -85,B 0,C 180,E1 -4228.777,E2 -4228.777} C_VEL
LIN {X 0,Y 655.904,Z 852.382,A -85,B 0,C 180,E1 -4230.699,E2 -4230.699} C_VEL
LIN {X 0,Y 655.911,Z 850.835,A -85,B 0,C 180,E1 -4232.709,E2 -4232.709} C_VEL
LIN {X 0,Y 655.924,Z 848.191,A -85,B 0,C 180,E1 -4234.371,E2 -4234.371} C_VEL
LIN {X 0,Y 655.948,Z 844.251,A -85,B 0,C 180,E1 -4236.037,E2 -4236.037} C_VEL
LIN {X 0,Y 655.99,Z 839.276,A -85,B 0,C 180,E1 -4237.62,E2 -4237.62} C_VEL
LIN {X 0,Y 656.11,Z 832.323,A -85,B 0,C 180,E1 -4239.385,E2 -4239.385} C_VEL
LIN {X 0,Y 656.327,Z 822.587,A -85,B 0,C 180,E1 -4241.334,E2 -4241.334} C_VEL
LIN {X 0,Y 656.604,Z 812.912,A -85,B 0,C 180,E1 -4242.935,E2 -4242.935} C_VEL
LIN {X 0,Y 656.952,Z 802.902,A -85,B 0,C 180,E1 -4244.364,E2 -4244.364} C_VEL
LIN {X 0,Y 657.396,Z 791.362,A -85,B 0,C 180,E1 -4245.799,E2 -4245.799} C_VEL
LIN {X 0,Y 658.061,Z 776.312,A -85,B 0,C 180,E1 -4247.417,E2 -4247.417} C_VEL
LIN {X 0,Y 658.776,Z 760.413,A -85,B 0,C 180,E1 -4248.862,E2 -4248.862} C_VEL
LIN {X 0,Y 659.421,Z 746.783,A -85,B 0,C 180,E1 -4249.948,E2 -4249.948} C_VEL
LIN {X 0,Y 660.109,Z 732.618,A -85,B 0,C 180,E1 -4250.945,E2 -4250.945} C_VEL
LIN {X 0,Y 660.808,Z 717.967,A -85,B 0,C 180,E1 -4251.853,E2 -4251.853} C_VEL
LIN {X 0,Y 661.452,Z 703.66,A -85,B 0,C 180,E1 -4252.631,E2 -4252.631} C_VEL
LIN {X 0,Y 662.067,Z 688.3,A -85,B 0,C 180,E1 -4253.356,E2 -4253.356} C_VEL
LIN {X 0,Y 662.768,Z 669.972,A -85,B 0,C 180,E1 -4254.085,E2 -4254.085} C_VEL
LIN {X 0,Y 663.459,Z 648.459,A -85,B 0,C 180,E1 -4254.776,E2 -4254.776} C_VEL
LIN {X 0,Y 663.992,Z 625.89,A -85,B 0,C 180,E1 -4255.314,E2 -4255.314} C_VEL
LIN {X 0,Y 664.319,Z 605.36,A -85,B 0,C 180,E1 -4255.653,E2 -4255.653} C_VEL
LIN {X 0,Y 667.251,Z 321.851,A -85,B 0,C 180,E1 -4259.039,E2 -4259.039} C_VEL
LIN {X 0,Y 665.89,Z 314.577,A -85,B 0,C 180,E1 -4259.21,E2 -4259.21} C_VEL
LIN {X 0,Y 666.879,Z 269.958,A -85,B 0,C 180,E1 -4262.362,E2 -4262.362} C_VEL
LIN {X 0,Y 668.183,Z 233.072,A -85,B 0,C 180,E1 -4265.093,E2 -4265.093} C_VEL
LIN {X 0,Y 661.541,Z 215.766,A -85,B 0,C 180,E1 -4266.767,E2 -4266.767} C_VEL
LIN {X 0,Y 656.721,Z 203.547,A -85,B 0,C 180,E1 -4267.879,E2 -4267.879} C_VEL
LIN {X 0,Y 656.677,Z 203.427,A -85,B 0,C 180,E1 -4270.954,E2 -4270.954} C_VEL
LIN {X 0,Y 656.703,Z 203.428,A -85,B 0,C 180,E1 -4273.972,E2 -4273.972} C_VEL
LIN {X 0,Y 656.68,Z 203.425,A -85,B 0,C 180,E1 -4276.988,E2 -4276.988} C_VEL
LIN {X 0,Y 656.699,Z 203.427,A -85,B 0,C 180,E1 -4279.984,E2 -4279.984} C_VEL
LIN {X 0,Y 656.683,Z 203.424,A -85,B 0,C 180,E1 -4283.071,E2 -4283.071} C_VEL
LIN {X 0,Y 656.696,Z 203.423,A -85,B 0,C 180,E1 -4286.08,E2 -4286.08} C_VEL
LIN {X 0,Y 656.687,Z 203.427,A -85,B 0,C 180,E1 -4289.128,E2 -4289.128} C_VEL
LIN {X 0,Y 656.694,Z 203.424,A -85,B 0,C 180,E1 -4292.131,E2 -4292.131} C_VEL
LIN {X 0,Y 656.69,Z 203.425,A -85,B 0,C 180,E1 -4295.16,E2 -4295.16} C_VEL
LIN {X 0,Y 656.692,Z 203.427,A -85,B 0,C 180,E1 -4298.191,E2 -4298.191} C_VEL
LIN {X 0,Y 656.693,Z 203.421,A -85,B 0,C 180,E1 -4301.26,E2 -4301.26} C_VEL
LIN {X 0,Y 656.687,Z 203.427,A -85,B 0,C 180,E1 -4304.274,E2 -4304.274} C_VEL
LIN {X 0,Y 656.695,Z 203.418,A -85,B 0,C 180,E1 -4307.245,E2 -4307.245} C_VEL
LIN {X 0,Y 656.685,Z 203.428,A -85,B 0,C 180,E1 -4310.27,E2 -4310.27} C_VEL
LIN {X 0,Y 656.697,Z 203.419,A -85,B 0,C 180,E1 -4313.267,E2 -4313.267} C_VEL
LIN {X 0,Y 656.682,Z 203.428,A -85,B 0,C 180,E1 -4316.333,E2 -4316.333} C_VEL
LIN {X 0,Y 656.698,Z 203.424,A -85,B 0,C 180,E1 -4319.389,E2 -4319.389} C_VEL
LIN {X 0,Y 656.677,Z 203.427,A -85,B 0,C 180,E1 -4322.356,E2 -4322.356} C_VEL
LIN {X 0,Y 656.701,Z 203.426,A -85,B 0,C 180,E1 -4325.417,E2 -4325.417} C_VEL
LIN {X 0,Y 656.674,Z 203.424,A -85,B 0,C 180,E1 -4328.405,E2 -4328.405} C_VEL
LIN {X 0,Y 656.703,Z 203.426,A -85,B 0,C 180,E1 -4331.416,E2 -4331.416} C_VEL
LIN {X 0,Y 656.671,Z 203.427,A -85,B 0,C 180,E1 -4334.461,E2 -4334.461} C_VEL
LIN {X 0,Y 656.706,Z 203.427,A -85,B 0,C 180,E1 -4337.455,E2 -4337.455} C_VEL
LIN {X 0,Y 656.669,Z 203.428,A -85,B 0,C 180,E1 -4340.501,E2 -4340.501} C_VEL
LIN {X 0,Y 656.708,Z 203.428,A -85,B 0,C 180,E1 -4343.511,E2 -4343.511} C_VEL
LIN {X 0,Y 656.665,Z 203.427,A -85,B 0,C 180,E1 -4346.497,E2 -4346.497} C_VEL
LIN {X 0,Y 656.711,Z 203.425,A -85,B 0,C 180,E1 -4349.459,E2 -4349.459} C_VEL
LIN {X 0,Y 656.661,Z 203.432,A -85,B 0,C 180,E1 -4352.514,E2 -4352.514} C_VEL
LIN {X 0,Y 656.708,Z 203.427,A -85,B 0,C 180,E1 -4355.458,E2 -4355.458} C_VEL
LIN {X 0,Y 656.658,Z 203.433,A -85,B 0,C 180,E1 -4358.52,E2 -4358.52} C_VEL
LIN {X 0,Y 656.713,Z 203.427,A -85,B 0,C 180,E1 -4361.487,E2 -4361.487} C_VEL
LIN {X 0,Y 656.655,Z 203.434,A -85,B 0,C 180,E1 -4364.551,E2 -4364.551} C_VEL
LIN {X 0,Y 656.733,Z 203.614,A -85,B 0,C 180,E1 -4365.91,E2 -4365.91} C_VEL
LIN {X 0,Y 657.964,Z 206.886,A -85,B 0,C 180,E1 -4366.207,E2 -4366.207} C_VEL
LIN {X 0,Y 666.705,Z 224.357,A -85,B 0,C 180,E1 -4367.935,E2 -4367.935} C_VEL
LIN {X 0,Y 673.617,Z 239.079,A -85,B 0,C 180,E1 -4369.257,E2 -4369.257} C_VEL
LIN {X 0,Y 671.5,Z 291.807,A -85,B 0,C 180,E1 -4371.888,E2 -4371.888} C_VEL
LIN {X 0,Y 671.164,Z 302.005,A -85,B 0,C 180,E1 -4372.375,E2 -4372.375} C_VEL
LIN {X 0,Y 673.391,Z 317.785,A -85,B 0,C 180,E1 -4372.716,E2 -4372.716} C_VEL
LIN {X 0,Y 671.173,Z 579.716,A -85,B 0,C 180,E1 -4375.827,E2 -4375.827} C_VEL
LIN {X 0,Y 670.199,Z 688.285,A -85,B 0,C 180,E1 -4377.108,E2 -4377.108} C_VEL
LIN {X 0,Y 669.641,Z 712.806,A -85,B 0,C 180,E1 -4377.524,E2 -4377.524} C_VEL
LIN {X 0,Y 668.783,Z 735.948,A -85,B 0,C 180,E1 -4378.076,E2 -4378.076} C_VEL
LIN {X 0,Y 667.921,Z 756.984,A -85,B 0,C 180,E1 -4378.704,E2 -4378.704} C_VEL
LIN {X 0,Y 666.738,Z 780.733,A -85,B 0,C 180,E1 -4379.578,E2 -4379.578} C_VEL
LIN {X 0,Y 665.734,Z 800.161,A -85,B 0,C 180,E1 -4380.432,E2 -4380.432} C_VEL
LIN {X 0,Y 664.477,Z 822.251,A -85,B 0,C 180,E1 -4381.558,E2 -4381.558} C_VEL
LIN {X 0,Y 663.221,Z 842.297,A -85,B 0,C 180,E1 -4382.755,E2 -4382.755} C_VEL
LIN {X 0,Y 662.03,Z 862.353,A -85,B 0,C 180,E1 -4384.12,E2 -4384.12} C_VEL
LIN {X 0,Y 660.824,Z 881.181,A -85,B 0,C 180,E1 -4385.602,E2 -4385.602} C_VEL
LIN {X 0,Y 659.791,Z 898.888,A -85,B 0,C 180,E1 -4387.172,E2 -4387.172} C_VEL
LIN {X 0,Y 658.834,Z 915.095,A -85,B 0,C 180,E1 -4388.826,E2 -4388.826} C_VEL
LIN {X 0,Y 658.029,Z 930.99,A -85,B 0,C 180,E1 -4390.655,E2 -4390.655} C_VEL
LIN {X 0,Y 657.344,Z 944.842,A -85,B 0,C 180,E1 -4392.504,E2 -4392.504} C_VEL
LIN {X 0,Y 656.828,Z 957.687,A -85,B 0,C 180,E1 -4394.459,E2 -4394.459} C_VEL
LIN {X 0,Y 656.443,Z 968.646,A -85,B 0,C 180,E1 -4396.434,E2 -4396.434} C_VEL
LIN {X 0,Y 656.206,Z 977.993,A -85,B 0,C 180,E1 -4398.397,E2 -4398.397} C_VEL
LIN {X 0,Y 656.049,Z 985.907,A -85,B 0,C 180,E1 -4400.437,E2 -4400.437} C_VEL
LIN {X 0,Y 655.943,Z 991.744,A -85,B 0,C 180,E1 -4402.291,E2 -4402.291} C_VEL
LIN {X 0,Y 655.912,Z 996.857,A -85,B 0,C 180,E1 -4404.401,E2 -4404.401} C_VEL
LIN {X 0,Y 655.914,Z 1000.012,A -85,B 0,C 180,E1 -4406.329,E2 -4406.329} C_VEL
LIN {X 0,Y 655.9,Z 1001.968,A -85,B 0,C 180,E1 -4408.34,E2 -4408.34} C_VEL
LIN {X 0,Y 655.885,Z 1002.395,A -85,B 0,C 180,E1 -4410.437,E2 -4410.437} C_VEL
LIN {X 0,Y 655.914,Z 1001.498,A -85,B 0,C 180,E1 -4412.272,E2 -4412.272} C_VEL
LIN {X 0,Y 655.92,Z 998.919,A -85,B 0,C 180,E1 -4414.462,E2 -4414.462} C_VEL
LIN {X 0,Y 655.93,Z 994.895,A -85,B 0,C 180,E1 -4416.477,E2 -4416.477} C_VEL
LIN {X 0,Y 655.985,Z 989.71,A -85,B 0,C 180,E1 -4418.414,E2 -4418.414} C_VEL
LIN {X 0,Y 656.122,Z 982.073,A -85,B 0,C 180,E1 -4420.597,E2 -4420.597} C_VEL
LIN {X 0,Y 656.307,Z 974.248,A -85,B 0,C 180,E1 -4422.426,E2 -4422.426} C_VEL
LIN {X 0,Y 656.637,Z 963.38,A -85,B 0,C 180,E1 -4424.552,E2 -4424.552} C_VEL
LIN {X 0,Y 657.027,Z 952.549,A -85,B 0,C 180,E1 -4426.352,E2 -4426.352} C_VEL
LIN {X 0,Y 657.641,Z 938.726,A -85,B 0,C 180,E1 -4428.344,E2 -4428.344} C_VEL
LIN {X 0,Y 658.309,Z 924.852,A -85,B 0,C 180,E1 -4430.076,E2 -4430.076} C_VEL
LIN {X 0,Y 659.245,Z 908.158,A -85,B 0,C 180,E1 -4431.908,E2 -4431.908} C_VEL
LIN {X 0,Y 660.181,Z 891.811,A -85,B 0,C 180,E1 -4433.474,E2 -4433.474} C_VEL
LIN {X 0,Y 661.369,Z 872.641,A -85,B 0,C 180,E1 -4435.095,E2 -4435.095} C_VEL
LIN {X 0,Y 662.48,Z 854.399,A -85,B 0,C 180,E1 -4436.439,E2 -4436.439} C_VEL
LIN {X 0,Y 663.804,Z 833.587,A -85,B 0,C 180,E1 -4437.788,E2 -4437.788} C_VEL
LIN {X 0,Y 664.99,Z 812.835,A -85,B 0,C 180,E1 -4438.942,E2 -4438.942} C_VEL
LIN {X 0,Y 666.28,Z 790.543,A -85,B 0,C 180,E1 -4440.013,E2 -4440.013} C_VEL
LIN {X 0,Y 667.346,Z 768.964,A -85,B 0,C 180,E1 -4440.875,E2 -4440.875} C_VEL
LIN {X 0,Y 668.306,Z 748.103,A -85,B 0,C 180,E1 -4441.578,E2 -4441.578} C_VEL
LIN {X 0,Y 669.246,Z 722.706,A -85,B 0,C 180,E1 -4442.257,E2 -4442.257} C_VEL
LIN {X 0,Y 669.926,Z 700.955,A -85,B 0,C 180,E1 -4442.695,E2 -4442.695} C_VEL
LIN {X 0,Y 670.482,Z 669.885,A -85,B 0,C 180,E1 -4443.127,E2 -4443.127} C_VEL
LIN {X 0,Y 671.201,Z 531.27,A -85,B 0,C 180,E1 -4444.678,E2 -4444.678} C_VEL
LIN {X 0,Y 671.916,Z 315.674,A -85,B 0,C 180,E1 -4447.099,E2 -4447.099} C_VEL
LIN {X 0,Y 669.934,Z 303.804,A -85,B 0,C 180,E1 -4447.347,E2 -4447.347} C_VEL
LIN {X 0,Y 671.509,Z 265.684,A -85,B 0,C 180,E1 -4449.26,E2 -4449.26} C_VEL
LIN {X 0,Y 673.601,Z 239.115,A -85,B 0,C 180,E1 -4450.73,E2 -4450.73} C_VEL
LIN {X 0,Y 668.998,Z 228.301,A -85,B 0,C 180,E1 -4451.92,E2 -4451.92} C_VEL
LIN {X 0,Y 665.749,Z 221.208,A -85,B 0,C 180,E1 -4452.872,E2 -4452.872} C_VEL
LIN {X 0,Y 663.628,Z 217.001,A -85,B 0,C 180,E1 -4453.554,E2 -4453.554} C_VEL
LIN {X 0,Y 661.75,Z 213.116,A -85,B 0,C 180,E1 -4454.273,E2 -4454.273} C_VEL
LIN {X 0,Y 659.752,Z 209.169,A -85,B 0,C 180,E1 -4455.176,E2 -4455.176} C_VEL
LIN {X 0,Y 657.358,Z 205.737,A -85,B 0,C 180,E1 -4456.515,E2 -4456.515} C_VEL
LIN {X 0,Y 656.751,Z 203.76,A -85,B 0,C 180,E1 -4457.725,E2 -4457.725} C_VEL
LIN {X 0,Y 656.789,Z 203.918,A -85,B 0,C 180,E1 -4458.769,E2 -4458.769} C_VEL
LIN {X 0,Y 657.572,Z 206.261,A -85,B 0,C 180,E1 -4460.029,E2 -4460.029} C_VEL
LIN {X 0,Y 659.559,Z 208.782,A -85,B 0,C 180,E1 -4461.051,E2 -4461.051} C_VEL
LIN {X 0,Y 661.234,Z 212.555,A -85,B 0,C 180,E1 -4461.905,E2 -4461.905} C_VEL
LIN {X 0,Y 662.091,Z 214.188,A -85,B 0,C 180,E1 -4462.241,E2 -4462.241} C_VEL
LIN {X 0,Y 663.998,Z 218.269,A -85,B 0,C 180,E1 -4462.962,E2 -4462.962} C_VEL
LIN {X 0,Y 667.432,Z 226.435,A -85,B 0,C 180,E1 -4464.143,E2 -4464.143} C_VEL
LIN {X 0,Y 670.543,Z 235.099,A -85,B 0,C 180,E1 -4465.172,E2 -4465.172} C_VEL
LIN {X 0,Y 667.26,Z 273.364,A -85,B 0,C 180,E1 -4467.76,E2 -4467.76} C_VEL
LIN {X 0,Y 664.493,Z 323.109,A -85,B 0,C 180,E1 -4470.92,E2 -4470.92} C_VEL
LIN {X 0,Y 662.644,Z 372.235,A -85,B 0,C 180,E1 -4473.905,E2 -4473.905} C_VEL
LIN {X 0,Y 661.052,Z 426.481,A -85,B 0,C 180,E1 -4477.096,E2 -4477.096} C_VEL
LIN {X 0,Y 660.499,Z 452.198,A -85,B 0,C 180,E1 -4478.562,E2 -4478.562} C_VEL
LIN {X 0,Y 664.049,Z 483.157,A -85,B 0,C 180,E1 -4479.228,E2 -4479.228} C_VEL
LIN {X 0,Y 661.565,Z 600.11,A -85,B 0,C 180,E1 -4480.849,E2 -4480.849} C_VEL
LIN {X 0,Y 660.467,Z 682.887,A -85,B 0,C 180,E1 -4481.945,E2 -4481.945} C_VEL
LIN {X 0,Y 660.109,Z 702.739,A -85,B 0,C 180,E1 -4482.368,E2 -4482.368} C_VEL
LIN {X 0,Y 659.696,Z 722.032,A -85,B 0,C 180,E1 -4482.945,E2 -4482.945} C_VEL
LIN {X 0,Y 659.228,Z 740.269,A -85,B 0,C 180,E1 -4483.659,E2 -4483.659} C_VEL
LIN {X 0,Y 658.773,Z 757.486,A -85,B 0,C 180,E1 -4484.506,E2 -4484.506} C_VEL
LIN {X 0,Y 658.3,Z 773.688,A -85,B 0,C 180,E1 -4485.486,E2 -4485.486} C_VEL
LIN {X 0,Y 657.845,Z 788.259,A -85,B 0,C 180,E1 -4486.553,E2 -4486.553} C_VEL
LIN {X 0,Y 657.43,Z 801.382,A -85,B 0,C 180,E1 -4487.706,E2 -4487.706} C_VEL
LIN {X 0,Y 657.065,Z 813.378,A -85,B 0,C 180,E1 -4488.972,E2 -4488.972} C_VEL
LIN {X 0,Y 656.748,Z 824.232,A -85,B 0,C 180,E1 -4490.359,E2 -4490.359} C_VEL
LIN {X 0,Y 656.503,Z 833.218,A -85,B 0,C 180,E1 -4491.769,E2 -4491.769} C_VEL
LIN {X 0,Y 656.333,Z 840.813,A -85,B 0,C 180,E1 -4493.263,E2 -4493.263} C_VEL
LIN {X 0,Y 656.229,Z 846.946,A -85,B 0,C 180,E1 -4494.842,E2 -4494.842} C_VEL
LIN {X 0,Y 656.142,Z 851.513,A -85,B 0,C 180,E1 -4496.505,E2 -4496.505} C_VEL
LIN {X 0,Y 656.102,Z 854.253,A -85,B 0,C 180,E1 -4498.166,E2 -4498.166} C_VEL
LIN {X 0,Y 656.085,Z 855.253,A -85,B 0,C 180,E1 -4499.825,E2 -4499.825} C_VEL
LIN {X 0,Y 656.073,Z 854.541,A -85,B 0,C 180,E1 -4501.485,E2 -4501.485} C_VEL
LIN {X 0,Y 656.091,Z 852.104,A -85,B 0,C 180,E1 -4503.145,E2 -4503.145} C_VEL
LIN {X 0,Y 656.129,Z 847.874,A -85,B 0,C 180,E1 -4504.808,E2 -4504.808} C_VEL
LIN {X 0,Y 656.21,Z 842.087,A -85,B 0,C 180,E1 -4506.386,E2 -4506.386} C_VEL
LIN {X 0,Y 656.349,Z 834.406,A -85,B 0,C 180,E1 -4507.969,E2 -4507.969} C_VEL
LIN {X 0,Y 656.569,Z 825.163,A -85,B 0,C 180,E1 -4509.467,E2 -4509.467} C_VEL
LIN {X 0,Y 656.862,Z 814.399,A -85,B 0,C 180,E1 -4510.88,E2 -4510.88} C_VEL
LIN {X 0,Y 657.227,Z 802.111,A -85,B 0,C 180,E1 -4512.209,E2 -4512.209} C_VEL
LIN {X 0,Y 657.662,Z 788.222,A -85,B 0,C 180,E1 -4513.451,E2 -4513.451} C_VEL
LIN {X 0,Y 658.121,Z 773.911,A -85,B 0,C 180,E1 -4514.518,E2 -4514.518} C_VEL
LIN {X 0,Y 658.613,Z 758.073,A -85,B 0,C 180,E1 -4515.498,E2 -4515.498} C_VEL
LIN {X 0,Y 659.072,Z 741.635,A -85,B 0,C 180,E1 -4516.332,E2 -4516.332} C_VEL
LIN {X 0,Y 659.568,Z 723.742,A -85,B 0,C 180,E1 -4517.058,E2 -4517.058} C_VEL
LIN {X 0,Y 659.981,Z 704.927,A -85,B 0,C 180,E1 -4517.644,E2 -4517.644} C_VEL
LIN {X 0,Y 660.339,Z 685.589,A -85,B 0,C 180,E1 -4518.075,E2 -4518.075} C_VEL
LIN {X 0,Y 660.619,Z 659.994,A -85,B 0,C 180,E1 -4518.426,E2 -4518.426} C_VEL
LIN {X 0,Y 662.276,Z 493.734,A -85,B 0,C 180,E1 -4520.426,E2 -4520.426} C_VEL
LIN {X 0,Y 661.35,Z 488.762,A -85,B 0,C 180,E1 -4520.523,E2 -4520.523} C_VEL
LIN {X 0,Y 654.524,Z 475.181,A -85,B 0,C 180,E1 -4520.955,E2 -4520.955} C_VEL
LIN {X 0,Y 653.858,Z 472.31,A -85,B 0,C 180,E1 -4521.017,E2 -4521.017} C_VEL
LIN {X 0,Y 652.75,Z 463.022,A -85,B 0,C 180,E1 -4521.193,E2 -4521.193} C_VEL
LIN {X 0,Y 654.174,Z 408.167,A -85,B 0,C 180,E1 -4524.374,E2 -4524.374} C_VEL
LIN {X 0,Y 655.734,Z 355.483,A -85,B 0,C 180,E1 -4527.474,E2 -4527.474} C_VEL
LIN {X 0,Y 657.428,Z 302.739,A -85,B 0,C 180,E1 -4530.631,E2 -4530.631} C_VEL
LIN {X 0,Y 659.179,Z 252.858,A -85,B 0,C 180,E1 -4533.671,E2 -4533.671} C_VEL
LIN {X 0,Y 659.907,Z 233.936,A -85,B 0,C 180,E1 -4534.836,E2 -4534.836} C_VEL
LIN {X 0,Y 650.721,Z 210.034,A -85,B 0,C 180,E1 -4536.928,E2 -4536.928} C_VEL
LIN {X 0,Y 648.77,Z 204.417,A -85,B 0,C 180,E1 -4537.431,E2 -4537.431} C_VEL
LIN {X 0,Y 648.696,Z 204.426,A -85,B 0,C 180,E1 -4540.461,E2 -4540.461} C_VEL
LIN {X 0,Y 648.771,Z 204.418,A -85,B 0,C 180,E1 -4543.455,E2 -4543.455} C_VEL
LIN {X 0,Y 648.761,Z 204.418,A -85,B 0,C 180,E1 -4546.576,E2 -4546.576} C_VEL
LIN {X 0,Y 648.778,Z 204.419,A -85,B 0,C 180,E1 -4549.72,E2 -4549.72} C_VEL
LIN {X 0,Y 648.766,Z 204.601,A -85,B 0,C 180,E1 -4551.755,E2 -4551.755} C_VEL
LIN {X 0,Y 651.485,Z 211.429,A -85,B 0,C 180,E1 -4552.369,E2 -4552.369} C_VEL
LIN {X 0,Y 659.281,Z 230.843,A -85,B 0,C 180,E1 -4554.234,E2 -4554.234} C_VEL
LIN {X 0,Y 661.28,Z 236.953,A -85,B 0,C 180,E1 -4554.824,E2 -4554.824} C_VEL
LIN {X 0,Y 659.905,Z 273.928,A -85,B 0,C 180,E1 -4557.562,E2 -4557.562} C_VEL
LIN {X 0,Y 659.196,Z 306.565,A -85,B 0,C 180,E1 -4559.863,E2 -4559.863} C_VEL
LIN {X 0,Y 659.229,Z 317.775,A -85,B 0,C 180,E1 -4560.601,E2 -4560.601} C_VEL
LIN {X 0,Y 660.287,Z 324.684,A -85,B 0,C 180,E1 -4560.741,E2 -4560.741} C_VEL
LIN {X 0,Y 657.859,Z 518.202,A -85,B 0,C 180,E1 -4563.114,E2 -4563.114} C_VEL
LIN {X 0,Y 656.758,Z 614.046,A -85,B 0,C 180,E1 -4564.306,E2 -4564.306} C_VEL
LIN {X 0,Y 656.299,Z 636.159,A -85,B 0,C 180,E1 -4564.745,E2 -4564.745} C_VEL
LIN {X 0,Y 655.685,Z 657.491,A -85,B 0,C 180,E1 -4565.33,E2 -4565.33} C_VEL
LIN {X 0,Y 655.003,Z 677.878,A -85,B 0,C 180,E1 -4566.042,E2 -4566.042} C_VEL
LIN {X 0,Y 654.138,Z 698.947,A -85,B 0,C 180,E1 -4566.964,E2 -4566.964} C_VEL
LIN {X 0,Y 653.28,Z 717.337,A -85,B 0,C 180,E1 -4567.943,E2 -4567.943} C_VEL
LIN {X 0,Y 652.47,Z 733.536,A -85,B 0,C 180,E1 -4568.952,E2 -4568.952} C_VEL
LIN {X 0,Y 651.674,Z 748.645,A -85,B 0,C 180,E1 -4570.038,E2 -4570.038} C_VEL
LIN {X 0,Y 650.748,Z 766.708,A -85,B 0,C 180,E1 -4571.547,E2 -4571.547} C_VEL
LIN {X 0,Y 650.053,Z 780.67,A -85,B 0,C 180,E1 -4572.915,E2 -4572.915} C_VEL
LIN {X 0,Y 649.515,Z 792.121,A -85,B 0,C 180,E1 -4574.188,E2 -4574.188} C_VEL
LIN {X 0,Y 649.06,Z 802.897,A -85,B 0,C 180,E1 -4575.548,E2 -4575.548} C_VEL
LIN {X 0,Y 648.693,Z 812.605,A -85,B 0,C 180,E1 -4576.948,E2 -4576.948} C_VEL
LIN {X 0,Y 648.408,Z 821.558,A -85,B 0,C 180,E1 -4578.436,E2 -4578.436} C_VEL
LIN {X 0,Y 648.172,Z 830.734,A -85,B 0,C 180,E1 -4580.23,E2 -4580.23} C_VEL
LIN {X 0,Y 648.011,Z 838.66,A -85,B 0,C 180,E1 -4582.196,E2 -4582.196} C_VEL
LIN {X 0,Y 647.956,Z 844,A -85,B 0,C 180,E1 -4583.888,E2 -4583.888} C_VEL
LIN {X 0,Y 647.925,Z 848.002,A -85,B 0,C 180,E1 -4585.575,E2 -4585.575} C_VEL
LIN {X 0,Y 647.91,Z 850.709,A -85,B 0,C 180,E1 -4587.258,E2 -4587.258} C_VEL
LIN {X 0,Y 647.912,Z 852.339,A -85,B 0,C 180,E1 -4589.204,E2 -4589.204} C_VEL
LIN {X 0,Y 647.901,Z 852.116,A -85,B 0,C 180,E1 -4591.238,E2 -4591.238} C_VEL
LIN {X 0,Y 647.905,Z 850.593,A -85,B 0,C 180,E1 -4592.919,E2 -4592.919} C_VEL
LIN {X 0,Y 647.924,Z 848.005,A -85,B 0,C 180,E1 -4594.514,E2 -4594.514} C_VEL
LIN {X 0,Y 647.958,Z 844.004,A -85,B 0,C 180,E1 -4596.201,E2 -4596.201} C_VEL
LIN {X 0,Y 648.01,Z 838.663,A -85,B 0,C 180,E1 -4597.893,E2 -4597.893} C_VEL
LIN {X 0,Y 648.173,Z 830.735,A -85,B 0,C 180,E1 -4599.859,E2 -4599.859} C_VEL
LIN {X 0,Y 648.408,Z 821.558,A -85,B 0,C 180,E1 -4601.655,E2 -4601.655} C_VEL
LIN {X 0,Y 648.679,Z 812.902,A -85,B 0,C 180,E1 -4603.096,E2 -4603.096} C_VEL
LIN {X 0,Y 649.035,Z 803.559,A -85,B 0,C 180,E1 -4604.452,E2 -4604.452} C_VEL
LIN {X 0,Y 649.481,Z 792.866,A -85,B 0,C 180,E1 -4605.813,E2 -4605.813} C_VEL
LIN {X 0,Y 650.008,Z 781.506,A -85,B 0,C 180,E1 -4607.086,E2 -4607.086} C_VEL
LIN {X 0,Y 650.637,Z 768.608,A -85,B 0,C 180,E1 -4608.363,E2 -4608.363} C_VEL
LIN {X 0,Y 651.548,Z 751.654,A -85,B 0,C 180,E1 -4609.825,E2 -4609.825} C_VEL
LIN {X 0,Y 652.411,Z 734.668,A -85,B 0,C 180,E1 -4611.063,E2 -4611.063} C_VEL
LIN {X 0,Y 653.221,Z 718.608,A -85,B 0,C 180,E1 -4612.073,E2 -4612.073} C_VEL
LIN {X 0,Y 653.96,Z 702.441,A -85,B 0,C 180,E1 -4612.948,E2 -4612.948} C_VEL
LIN {X 0,Y 654.802,Z 683.002,A -85,B 0,C 180,E1 -4613.839,E2 -4613.839} C_VEL
LIN {X 0,Y 655.55,Z 661.856,A -85,B 0,C 180,E1 -4614.623,E2 -4614.623} C_VEL
LIN {X 0,Y 656.187,Z 640.976,A -85,B 0,C 180,E1 -4615.229,E2 -4615.229} C_VEL
LIN {X 0,Y 656.632,Z 619.434,A -85,B 0,C 180,E1 -4615.687,E2 -4615.687} C_VEL
LIN {X 0,Y 657.002,Z 593.281,A -85,B 0,C 180,E1 -4616.058,E2 -4616.058} C_VEL
LIN {X 0,Y 660.174,Z 335.018,A -85,B 0,C 180,E1 -4619.227,E2 -4619.227} C_VEL
LIN {X 0,Y 660.114,Z 322.291,A -85,B 0,C 180,E1 -4619.389,E2 -4619.389} C_VEL
LIN {X 0,Y 659.163,Z 317.144,A -85,B 0,C 180,E1 -4619.513,E2 -4619.513} C_VEL
LIN {X 0,Y 659.693,Z 280.043,A -85,B 0,C 180,E1 -4622.083,E2 -4622.083} C_VEL
LIN {X 0,Y 661.162,Z 241.324,A -85,B 0,C 180,E1 -4624.947,E2 -4624.947} C_VEL
LIN {X 0,Y 661.205,Z 236.237,A -85,B 0,C 180,E1 -4625.328,E2 -4625.328} C_VEL
LIN {X 0,Y 654.289,Z 218.189,A -85,B 0,C 180,E1 -4627.086,E2 -4627.086} C_VEL
LIN {X 0,Y 648.793,Z 204.584,A -85,B 0,C 180,E1 -4628.344,E2 -4628.344} C_VEL
LIN {X 0,Y 648.748,Z 204.415,A -85,B 0,C 180,E1 -4631.392,E2 -4631.392} C_VEL
LIN {X 0,Y 648.762,Z 204.418,A -85,B 0,C 180,E1 -4634.598,E2 -4634.598} C_VEL
LIN {X 0,Y 648.769,Z 204.424,A -85,B 0,C 180,E1 -4637.781,E2 -4637.781} C_VEL
LIN {X 0,Y 648.748,Z 204.416,A -85,B 0,C 180,E1 -4640.922,E2 -4640.922} C_VEL
LIN {X 0,Y 648.761,Z 204.417,A -85,B 0,C 180,E1 -4644.013,E2 -4644.013} C_VEL
LIN {X 0,Y 648.748,Z 204.408,A -85,B 0,C 180,E1 -4647.039,E2 -4647.039} C_VEL
LIN {X 0,Y 648.757,Z 204.414,A -85,B 0,C 180,E1 -4650.042,E2 -4650.042} C_VEL
LIN {X 0,Y 648.753,Z 204.411,A -85,B 0,C 180,E1 -4653.055,E2 -4653.055} C_VEL
LIN {X 0,Y 648.755,Z 204.403,A -85,B 0,C 180,E1 -4656.087,E2 -4656.087} C_VEL
LIN {X 0,Y 648.754,Z 204.414,A -85,B 0,C 180,E1 -4659.143,E2 -4659.143} C_VEL
LIN {X 0,Y 648.752,Z 204.405,A -85,B 0,C 180,E1 -4662.139,E2 -4662.139} C_VEL
LIN {X 0,Y 648.757,Z 204.413,A -85,B 0,C 180,E1 -4665.176,E2 -4665.176} C_VEL
LIN {X 0,Y 648.746,Z 204.408,A -85,B 0,C 180,E1 -4668.261,E2 -4668.261} C_VEL
LIN {X 0,Y 648.758,Z 204.416,A -85,B 0,C 180,E1 -4671.313,E2 -4671.313} C_VEL
LIN {X 0,Y 648.742,Z 204.405,A -85,B 0,C 180,E1 -4674.339,E2 -4674.339} C_VEL
LIN {X 0,Y 648.76,Z 204.417,A -85,B 0,C 180,E1 -4677.438,E2 -4677.438} C_VEL
LIN {X 0,Y 648.738,Z 204.399,A -85,B 0,C 180,E1 -4680.442,E2 -4680.442} C_VEL
LIN {X 0,Y 648.763,Z 204.416,A -85,B 0,C 180,E1 -4683.534,E2 -4683.534} C_VEL
LIN {X 0,Y 648.736,Z 204.4,A -85,B 0,C 180,E1 -4686.549,E2 -4686.549} C_VEL
LIN {X 0,Y 648.765,Z 204.414,A -85,B 0,C 180,E1 -4689.582,E2 -4689.582} C_VEL
LIN {X 0,Y 648.735,Z 204.415,A -85,B 0,C 180,E1 -4692.642,E2 -4692.642} C_VEL
LIN {X 0,Y 648.77,Z 204.416,A -85,B 0,C 180,E1 -4695.739,E2 -4695.739} C_VEL
LIN {X 0,Y 648.735,Z 204.413,A -85,B 0,C 180,E1 -4698.792,E2 -4698.792} C_VEL
LIN {X 0,Y 648.769,Z 204.417,A -85,B 0,C 180,E1 -4701.904,E2 -4701.904} C_VEL
LIN {X 0,Y 648.742,Z 204.415,A -85,B 0,C 180,E1 -4704.981,E2 -4704.981} C_VEL
LIN {X 0,Y 648.738,Z 204.42,A -85,B 0,C 180,E1 -4708.241,E2 -4708.241} C_VEL
LIN {X 0,Y 648.754,Z 204.415,A -85,B 0,C 180,E1 -4711.197,E2 -4711.197} C_VEL
LIN {X 0,Y 648.73,Z 204.422,A -85,B 0,C 180,E1 -4714.341,E2 -4714.341} C_VEL
LIN {X 0,Y 648.759,Z 204.416,A -85,B 0,C 180,E1 -4717.319,E2 -4717.319} C_VEL
LIN {X 0,Y 648.722,Z 204.424,A -85,B 0,C 180,E1 -4720.459,E2 -4720.459} C_VEL
LIN {X 0,Y 648.764,Z 204.415,A -85,B 0,C 180,E1 -4723.455,E2 -4723.455} C_VEL
LIN {X 0,Y 648.754,Z 204.491,A -85,B 0,C 180,E1 -4725.291,E2 -4725.291} C_VEL
LIN {X 0,Y 649.81,Z 207.478,A -85,B 0,C 180,E1 -4725.563,E2 -4725.563} C_VEL
LIN {X 0,Y 651.127,Z 209.868,A -85,B 0,C 180,E1 -4725.819,E2 -4725.819} C_VEL
LIN {X 0,Y 660.682,Z 229.107,A -85,B 0,C 180,E1 -4727.737,E2 -4727.737} C_VEL
LIN {X 0,Y 667.072,Z 242.765,A -85,B 0,C 180,E1 -4728.982,E2 -4728.982} C_VEL
LIN {X 0,Y 664.694,Z 294.604,A -85,B 0,C 180,E1 -4731.604,E2 -4731.604} C_VEL
LIN {X 0,Y 664.435,Z 302.698,A -85,B 0,C 180,E1 -4731.99,E2 -4731.99} C_VEL
LIN {X 0,Y 666.726,Z 319.035,A -85,B 0,C 180,E1 -4732.348,E2 -4732.348} C_VEL
LIN {X 0,Y 664.185,Z 578.073,A -85,B 0,C 180,E1 -4735.473,E2 -4735.473} C_VEL
LIN {X 0,Y 663.137,Z 691.841,A -85,B 0,C 180,E1 -4736.825,E2 -4736.825} C_VEL
LIN {X 0,Y 662.495,Z 717.649,A -85,B 0,C 180,E1 -4737.285,E2 -4737.285} C_VEL
LIN {X 0,Y 661.775,Z 739.01,A -85,B 0,C 180,E1 -4737.796,E2 -4737.796} C_VEL
LIN {X 0,Y 660.812,Z 761.255,A -85,B 0,C 180,E1 -4738.481,E2 -4738.481} C_VEL
LIN {X 0,Y 659.599,Z 783.335,A -85,B 0,C 180,E1 -4739.329,E2 -4739.329} C_VEL
LIN {X 0,Y 658.38,Z 805.273,A -85,B 0,C 180,E1 -4740.324,E2 -4740.324} C_VEL
LIN {X 0,Y 656.935,Z 827.118,A -85,B 0,C 180,E1 -4741.5,E2 -4741.5} C_VEL
LIN {X 0,Y 655.618,Z 847.65,A -85,B 0,C 180,E1 -4742.772,E2 -4742.772} C_VEL
LIN {X 0,Y 654.267,Z 867.218,A -85,B 0,C 180,E1 -4744.179,E2 -4744.179} C_VEL
LIN {X 0,Y 653.067,Z 885.201,A -85,B 0,C 180,E1 -4745.643,E2 -4745.643} C_VEL
LIN {X 0,Y 651.923,Z 902.603,A -85,B 0,C 180,E1 -4747.263,E2 -4747.263} C_VEL
LIN {X 0,Y 650.986,Z 917.629,A -85,B 0,C 180,E1 -4748.841,E2 -4748.841} C_VEL
LIN {X 0,Y 650.064,Z 934.017,A -85,B 0,C 180,E1 -4750.808,E2 -4750.808} C_VEL
LIN {X 0,Y 649.404,Z 947.155,A -85,B 0,C 180,E1 -4752.62,E2 -4752.62} C_VEL
LIN {X 0,Y 648.818,Z 960.384,A -85,B 0,C 180,E1 -4754.738,E2 -4754.738} C_VEL
LIN {X 0,Y 648.459,Z 970.021,A -85,B 0,C 180,E1 -4756.536,E2 -4756.536} C_VEL
LIN {X 0,Y 648.175,Z 979.834,A -85,B 0,C 180,E1 -4758.702,E2 -4758.702} C_VEL
LIN {X 0,Y 648.054,Z 986.817,A -85,B 0,C 180,E1 -4760.587,E2 -4760.587} C_VEL
LIN {X 0,Y 647.946,Z 993.244,A -85,B 0,C 180,E1 -4762.73,E2 -4762.73} C_VEL
LIN {X 0,Y 647.896,Z 997.656,A -85,B 0,C 180,E1 -4764.776,E2 -4764.776} C_VEL
LIN {X 0,Y 647.904,Z 1000.463,A -85,B 0,C 180,E1 -4766.638,E2 -4766.638} C_VEL
LIN {X 0,Y 647.909,Z 1002.215,A -85,B 0,C 180,E1 -4768.85,E2 -4768.85} C_VEL
LIN {X 0,Y 647.885,Z 1002.328,A -85,B 0,C 180,E1 -4770.707,E2 -4770.707} C_VEL
LIN {X 0,Y 647.888,Z 1001.225,A -85,B 0,C 180,E1 -4772.654,E2 -4772.654} C_VEL
LIN {X 0,Y 647.903,Z 998.291,A -85,B 0,C 180,E1 -4774.869,E2 -4774.869} C_VEL
LIN {X 0,Y 647.937,Z 994.689,A -85,B 0,C 180,E1 -4776.646,E2 -4776.646} C_VEL
LIN {X 0,Y 647.991,Z 989.202,A -85,B 0,C 180,E1 -4778.698,E2 -4778.698} C_VEL
LIN {X 0,Y 648.14,Z 981.956,A -85,B 0,C 180,E1 -4780.758,E2 -4780.758} C_VEL
LIN {X 0,Y 648.361,Z 973.937,A -85,B 0,C 180,E1 -4782.65,E2 -4782.65} C_VEL
LIN {X 0,Y 648.736,Z 962.864,A -85,B 0,C 180,E1 -4784.824,E2 -4784.824} C_VEL
LIN {X 0,Y 649.179,Z 951.908,A -85,B 0,C 180,E1 -4786.658,E2 -4786.658} C_VEL
LIN {X 0,Y 649.881,Z 937.323,A -85,B 0,C 180,E1 -4788.758,E2 -4788.758} C_VEL
LIN {X 0,Y 650.669,Z 923.308,A -85,B 0,C 180,E1 -4790.51,E2 -4790.51} C_VEL
LIN {X 0,Y 651.685,Z 906.306,A -85,B 0,C 180,E1 -4792.365,E2 -4792.365} C_VEL
LIN {X 0,Y 652.725,Z 890.29,A -85,B 0,C 180,E1 -4793.902,E2 -4793.902} C_VEL
LIN {X 0,Y 654.04,Z 870.36,A -85,B 0,C 180,E1 -4795.579,E2 -4795.579} C_VEL
LIN {X 0,Y 655.281,Z 852.393,A -85,B 0,C 180,E1 -4796.9,E2 -4796.9} C_VEL
LIN {X 0,Y 656.73,Z 830.354,A -85,B 0,C 180,E1 -4798.312,E2 -4798.312} C_VEL
LIN {X 0,Y 657.987,Z 810.743,A -85,B 0,C 180,E1 -4799.396,E2 -4799.396} C_VEL
LIN {X 0,Y 659.434,Z 786.726,A -85,B 0,C 180,E1 -4800.528,E2 -4800.528} C_VEL
LIN {X 0,Y 660.465,Z 767.674,A -85,B 0,C 180,E1 -4801.284,E2 -4801.284} C_VEL
LIN {X 0,Y 661.518,Z 746.017,A -85,B 0,C 180,E1 -4802.009,E2 -4802.009} C_VEL
LIN {X 0,Y 662.289,Z 722.664,A -85,B 0,C 180,E1 -4802.604,E2 -4802.604} C_VEL
LIN {X 0,Y 662.833,Z 700.466,A -85,B 0,C 180,E1 -4803.022,E2 -4803.022} C_VEL
LIN {X 0,Y 663.226,Z 667.583,A -85,B 0,C 180,E1 -4803.441,E2 -4803.441} C_VEL
LIN {X 0,Y 664.223,Z 431.13,A -85,B 0,C 180,E1 -4806.075,E2 -4806.075} C_VEL
LIN {X 0,Y 664.615,Z 316.21,A -85,B 0,C 180,E1 -4807.405,E2 -4807.405} C_VEL
LIN {X 0,Y 662.885,Z 306.048,A -85,B 0,C 180,E1 -4807.614,E2 -4807.614} C_VEL
LIN {X 0,Y 664.642,Z 271.267,A -85,B 0,C 180,E1 -4809.41,E2 -4809.41} C_VEL
LIN {X 0,Y 667.165,Z 243.082,A -85,B 0,C 180,E1 -4811.009,E2 -4811.009} C_VEL
LIN {X 0,Y 663.154,Z 233.195,A -85,B 0,C 180,E1 -4812.141,E2 -4812.141} C_VEL
LIN {X 0,Y 660.075,Z 226.378,A -85,B 0,C 180,E1 -4813.102,E2 -4813.102} C_VEL
LIN {X 0,Y 658.312,Z 222.717,A -85,B 0,C 180,E1 -4813.716,E2 -4813.716} C_VEL
LIN {X 0,Y 656.59,Z 219.08,A -85,B 0,C 180,E1 -4814.421,E2 -4814.421} C_VEL
LIN {X 0,Y 654.484,Z 214.797,A -85,B 0,C 180,E1 -4815.473,E2 -4815.473} C_VEL
LIN {X 0,Y 652.478,Z 211.672,A -85,B 0,C 180,E1 -4816.84,E2 -4816.84} C_VEL
LIN {X 0,Y 652.161,Z 210.241,A -85,B 0,C 180,E1 -4817.932,E2 -4817.932} C_VEL
LIN {X 0,Y 652.217,Z 210.604,A -85,B 0,C 180,E1 -4818.876,E2 -4818.876} C_VEL
LIN {X 0,Y 653.16,Z 213.211,A -85,B 0,C 180,E1 -4820.218,E2 -4820.218} C_VEL
LIN {X 0,Y 654.639,Z 215.367,A -85,B 0,C 180,E1 -4821.027,E2 -4821.027} C_VEL
LIN {X 0,Y 656.516,Z 219.112,A -85,B 0,C 180,E1 -4821.944,E2 -4821.944} C_VEL
LIN {X 0,Y 659.162,Z 225.507,A -85,B 0,C 180,E1 -4823.08,E2 -4823.08} C_VEL
LIN {X 0,Y 662.192,Z 233.136,A -85,B 0,C 180,E1 -4824.18,E2 -4824.18} C_VEL
LIN {X 0,Y 664.172,Z 238.986,A -85,B 0,C 180,E1 -4824.894,E2 -4824.894} C_VEL
LIN {X 0,Y 660.624,Z 275.053,A -85,B 0,C 180,E1 -4827.396,E2 -4827.396} C_VEL
LIN {X 0,Y 657.552,Z 322.58,A -85,B 0,C 180,E1 -4830.483,E2 -4830.483} C_VEL
LIN {X 0,Y 655.519,Z 368.995,A -85,B 0,C 180,E1 -4833.361,E2 -4833.361} C_VEL
LIN {X 0,Y 653.654,Z 424.889,A -85,B 0,C 180,E1 -4836.707,E2 -4836.707} C_VEL
LIN {X 0,Y 653.059,Z 449.561,A -85,B 0,C 180,E1 -4838.128,E2 -4838.128} C_VEL
LIN {X 0,Y 656.988,Z 483.372,A -85,B 0,C 180,E1 -4838.902,E2 -4838.902} C_VEL
LIN {X 0,Y 654.028,Z 608.597,A -85,B 0,C 180,E1 -4840.696,E2 -4840.696} C_VEL
LIN {X 0,Y 652.919,Z 683.38,A -85,B 0,C 180,E1 -4841.718,E2 -4841.718} C_VEL
LIN {X 0,Y 652.51,Z 703.626,A -85,B 0,C 180,E1 -4842.162,E2 -4842.162} C_VEL
LIN {X 0,Y 652.068,Z 722.573,A -85,B 0,C 180,E1 -4842.739,E2 -4842.739} C_VEL
LIN {X 0,Y 651.536,Z 741.817,A -85,B 0,C 180,E1 -4843.506,E2 -4843.506} C_VEL
LIN {X 0,Y 651.061,Z 758.714,A -85,B 0,C 180,E1 -4844.353,E2 -4844.353} C_VEL
LIN {X 0,Y 650.555,Z 774.907,A -85,B 0,C 180,E1 -4845.346,E2 -4845.346} C_VEL
LIN {X 0,Y 650.067,Z 789.577,A -85,B 0,C 180,E1 -4846.434,E2 -4846.434} C_VEL
LIN {X 0,Y 649.64,Z 802.211,A -85,B 0,C 180,E1 -4847.556,E2 -4847.556} C_VEL
LIN {X 0,Y 649.249,Z 814.143,A -85,B 0,C 180,E1 -4848.821,E2 -4848.821} C_VEL
LIN {X 0,Y 648.901,Z 825.187,A -85,B 0,C 180,E1 -4850.241,E2 -4850.241} C_VEL
LIN {X 0,Y 648.634,Z 834.216,A -85,B 0,C 180,E1 -4851.668,E2 -4851.668} C_VEL
LIN {X 0,Y 648.438,Z 842.116,A -85,B 0,C 180,E1 -4853.241,E2 -4853.241} C_VEL
LIN {X 0,Y 648.319,Z 848.304,A -85,B 0,C 180,E1 -4854.868,E2 -4854.868} C_VEL
LIN {X 0,Y 648.225,Z 852.586,A -85,B 0,C 180,E1 -4856.463,E2 -4856.463} C_VEL
LIN {X 0,Y 648.176,Z 855.317,A -85,B 0,C 180,E1 -4858.144,E2 -4858.144} C_VEL
LIN {X 0,Y 648.153,Z 856.294,A -85,B 0,C 180,E1 -4859.823,E2 -4859.823} C_VEL
LIN {X 0,Y 648.138,Z 855.546,A -85,B 0,C 180,E1 -4861.503,E2 -4861.503} C_VEL
LIN {X 0,Y 648.156,Z 853.062,A -85,B 0,C 180,E1 -4863.184,E2 -4863.184} C_VEL
LIN {X 0,Y 648.196,Z 849,A -85,B 0,C 180,E1 -4864.791,E2 -4864.791} C_VEL
LIN {X 0,Y 648.282,Z 843.29,A -85,B 0,C 180,E1 -4866.376,E2 -4866.376} C_VEL
LIN {X 0,Y 648.429,Z 835.65,A -85,B 0,C 180,E1 -4867.977,E2 -4867.977} C_VEL
LIN {X 0,Y 648.665,Z 826.463,A -85,B 0,C 180,E1 -4869.494,E2 -4869.494} C_VEL
LIN {X 0,Y 648.978,Z 815.776,A -85,B 0,C 180,E1 -4870.924,E2 -4870.924} C_VEL
LIN {X 0,Y 649.367,Z 803.582,A -85,B 0,C 180,E1 -4872.268,E2 -4872.268} C_VEL
LIN {X 0,Y 649.833,Z 789.819,A -85,B 0,C 180,E1 -4873.526,E2 -4873.526} C_VEL
LIN {X 0,Y 650.339,Z 774.993,A -85,B 0,C 180,E1 -4874.65,E2 -4874.65} C_VEL
LIN {X 0,Y 650.865,Z 759.237,A -85,B 0,C 180,E1 -4875.641,E2 -4875.641} C_VEL
LIN {X 0,Y 651.383,Z 741.984,A -85,B 0,C 180,E1 -4876.528,E2 -4876.528} C_VEL
LIN {X 0,Y 651.915,Z 724,A -85,B 0,C 180,E1 -4877.265,E2 -4877.265} C_VEL
LIN {X 0,Y 652.363,Z 705.072,A -85,B 0,C 180,E1 -4877.861,E2 -4877.861} C_VEL
LIN {X 0,Y 652.749,Z 685.577,A -85,B 0,C 180,E1 -4878.299,E2 -4878.299} C_VEL
LIN {X 0,Y 653.055,Z 660.087,A -85,B 0,C 180,E1 -4878.653,E2 -4878.653} C_VEL
LIN {X 0,Y 654.97,Z 481.489,A -85,B 0,C 180,E1 -4880.855,E2 -4880.855} C_VEL
LIN {X 0,Y 653.858,Z 472.31,A -85,B 0,C 180,E1 -4881.017,E2 -4881.017} C_VEL
LIN {X 0,Y 652.368,Z 467.523,A -85,B 0,C 180,E1 -4881.156,E2 -4881.156} C_VEL
LIN {X 0,Y 648.117,Z 460.613,A -85,B 0,C 180,E1 -4881.537,E2 -4881.537} C_VEL
LIN {X 0,Y 645.709,Z 455.501,A -85,B 0,C 180,E1 -4881.882,E2 -4881.882} C_VEL
LIN {X 0,Y 645.421,Z 453.034,A -85,B 0,C 180,E1 -4882.035,E2 -4882.035} C_VEL
LIN {X 0,Y 646.89,Z 401.363,A -85,B 0,C 180,E1 -4885.072,E2 -4885.072} C_VEL
LIN {X 0,Y 648.629,Z 348.941,A -85,B 0,C 180,E1 -4888.196,E2 -4888.196} C_VEL
LIN {X 0,Y 650.482,Z 295.296,A -85,B 0,C 180,E1 -4891.447,E2 -4891.447} C_VEL
LIN {X 0,Y 652.355,Z 247.523,A -85,B 0,C 180,E1 -4894.39,E2 -4894.39} C_VEL
LIN {X 0,Y 652.743,Z 236.826,A -85,B 0,C 180,E1 -4895.06,E2 -4895.06} C_VEL
LIN {X 0,Y 643.253,Z 211.934,A -85,B 0,C 180,E1 -4897.263,E2 -4897.263} C_VEL
LIN {X 0,Y 640.828,Z 205.41,A -85,B 0,C 180,E1 -4897.859,E2 -4897.859} C_VEL
LIN {X 0,Y 640.773,Z 205.416,A -85,B 0,C 180,E1 -4900.831,E2 -4900.831} C_VEL
LIN {X 0,Y 640.8,Z 205.409,A -85,B 0,C 180,E1 -4904,E2 -4904} C_VEL
LIN {X 0,Y 640.808,Z 205.405,A -85,B 0,C 180,E1 -4907.009,E2 -4907.009} C_VEL
LIN {X 0,Y 640.791,Z 205.412,A -85,B 0,C 180,E1 -4910.15,E2 -4910.15} C_VEL
LIN {X 0,Y 640.821,Z 205.644,A -85,B 0,C 180,E1 -4911.276,E2 -4911.276} C_VEL
LIN {X 0,Y 649.199,Z 226.246,A -85,B 0,C 180,E1 -4913.216,E2 -4913.216} C_VEL
LIN {X 0,Y 654.391,Z 240.008,A -85,B 0,C 180,E1 -4914.582,E2 -4914.582} C_VEL
LIN {X 0,Y 653.041,Z 276.512,A -85,B 0,C 180,E1 -4917.283,E2 -4917.283} C_VEL
LIN {X 0,Y 652.349,Z 308.899,A -85,B 0,C 180,E1 -4919.564,E2 -4919.564} C_VEL
LIN {X 0,Y 652.483,Z 320.092,A -85,B 0,C 180,E1 -4920.284,E2 -4920.284} C_VEL
LIN {X 0,Y 653.351,Z 326.024,A -85,B 0,C 180,E1 -4920.405,E2 -4920.405} C_VEL
LIN {X 0,Y 651.375,Z 465.842,A -85,B 0,C 180,E1 -4922.146,E2 -4922.146} C_VEL
LIN {X 0,Y 649.238,Z 615.863,A -85,B 0,C 180,E1 -4924.085,E2 -4924.085} C_VEL
LIN {X 0,Y 648.756,Z 638.263,A -85,B 0,C 180,E1 -4924.545,E2 -4924.545} C_VEL
LIN {X 0,Y 648.087,Z 660.194,A -85,B 0,C 180,E1 -4925.163,E2 -4925.163} C_VEL
LIN {X 0,Y 647.338,Z 681.426,A -85,B 0,C 180,E1 -4925.935,E2 -4925.935} C_VEL
LIN {X 0,Y 646.5,Z 701.268,A -85,B 0,C 180,E1 -4926.82,E2 -4926.82} C_VEL
LIN {X 0,Y 645.592,Z 720.156,A -85,B 0,C 180,E1 -4927.848,E2 -4927.848} C_VEL
LIN {X 0,Y 644.604,Z 738.54,A -85,B 0,C 180,E1 -4929.037,E2 -4929.037} C_VEL
LIN {X 0,Y 643.611,Z 756.559,A -85,B 0,C 180,E1 -4930.419,E2 -4930.419} C_VEL
LIN {X 0,Y 642.804,Z 770.655,A -85,B 0,C 180,E1 -4931.687,E2 -4931.687} C_VEL
LIN {X 0,Y 642.12,Z 783.236,A -85,B 0,C 180,E1 -4932.977,E2 -4932.977} C_VEL
LIN {X 0,Y 641.566,Z 794.393,A -85,B 0,C 180,E1 -4934.265,E2 -4934.265} C_VEL
LIN {X 0,Y 641.041,Z 806.241,A -85,B 0,C 180,E1 -4935.825,E2 -4935.825} C_VEL
LIN {X 0,Y 640.558,Z 818.494,A -85,B 0,C 180,E1 -4937.743,E2 -4937.743} C_VEL
LIN {X 0,Y 640.296,Z 827.228,A -85,B 0,C 180,E1 -4939.381,E2 -4939.381} C_VEL
LIN {X 0,Y 640.119,Z 834.156,A -85,B 0,C 180,E1 -4940.923,E2 -4940.923} C_VEL
LIN {X 0,Y 640.003,Z 839.874,A -85,B 0,C 180,E1 -4942.459,E2 -4942.459} C_VEL
LIN {X 0,Y 639.952,Z 844.477,A -85,B 0,C 180,E1 -4943.991,E2 -4943.991} C_VEL
LIN {X 0,Y 639.927,Z 848.355,A -85,B 0,C 180,E1 -4945.699,E2 -4945.699} C_VEL
LIN {X 0,Y 639.912,Z 851.284,A -85,B 0,C 180,E1 -4947.672,E2 -4947.672} C_VEL
LIN {X 0,Y 639.904,Z 852.406,A -85,B 0,C 180,E1 -4949.731,E2 -4949.731} C_VEL
LIN {X 0,Y 639.898,Z 851.993,A -85,B 0,C 180,E1 -4951.433,E2 -4951.433} C_VEL
LIN {X 0,Y 639.902,Z 850.469,A -85,B 0,C 180,E1 -4953.045,E2 -4953.045} C_VEL
LIN {X 0,Y 639.921,Z 847.819,A -85,B 0,C 180,E1 -4954.66,E2 -4954.66} C_VEL
LIN {X 0,Y 639.963,Z 843.997,A -85,B 0,C 180,E1 -4956.279,E2 -4956.279} C_VEL
LIN {X 0,Y 640.025,Z 838.659,A -85,B 0,C 180,E1 -4957.992,E2 -4957.992} C_VEL
LIN {X 0,Y 640.203,Z 830.73,A -85,B 0,C 180,E1 -4959.983,E2 -4959.983} C_VEL
LIN {X 0,Y 640.459,Z 821.549,A -85,B 0,C 180,E1 -4961.801,E2 -4961.801} C_VEL
LIN {X 0,Y 640.761,Z 812.893,A -85,B 0,C 180,E1 -4963.261,E2 -4963.261} C_VEL
LIN {X 0,Y 641.147,Z 803.547,A -85,B 0,C 180,E1 -4964.634,E2 -4964.634} C_VEL
LIN {X 0,Y 641.609,Z 793.434,A -85,B 0,C 180,E1 -4965.941,E2 -4965.941} C_VEL
LIN {X 0,Y 642.168,Z 782.351,A -85,B 0,C 180,E1 -4967.208,E2 -4967.208} C_VEL
LIN {X 0,Y 642.858,Z 769.665,A -85,B 0,C 180,E1 -4968.5,E2 -4968.5} C_VEL
LIN {X 0,Y 643.734,Z 754.551,A -85,B 0,C 180,E1 -4969.84,E2 -4969.84} C_VEL
LIN {X 0,Y 644.709,Z 736.664,A -85,B 0,C 180,E1 -4971.184,E2 -4971.184} C_VEL
LIN {X 0,Y 645.707,Z 717.565,A -85,B 0,C 180,E1 -4972.392,E2 -4972.392} C_VEL
LIN {X 0,Y 646.617,Z 698.841,A -85,B 0,C 180,E1 -4973.388,E2 -4973.388} C_VEL
LIN {X 0,Y 647.437,Z 678.959,A -85,B 0,C 180,E1 -4974.255,E2 -4974.255} C_VEL
LIN {X 0,Y 648.111,Z 659.134,A -85,B 0,C 180,E1 -4974.958,E2 -4974.958} C_VEL
LIN {X 0,Y 648.75,Z 638.223,A -85,B 0,C 180,E1 -4975.544,E2 -4975.544} C_VEL
LIN {X 0,Y 649.218,Z 616.481,A -85,B 0,C 180,E1 -4975.994,E2 -4975.994} C_VEL
LIN {X 0,Y 649.909,Z 565.175,A -85,B 0,C 180,E1 -4976.67,E2 -4976.67} C_VEL
LIN {X 0,Y 652.937,Z 359.404,A -85,B 0,C 180,E1 -4979.282,E2 -4979.282} C_VEL
LIN {X 0,Y 653.179,Z 323.688,A -85,B 0,C 180,E1 -4979.724,E2 -4979.724} C_VEL
LIN {X 0,Y 652.385,Z 319.37,A -85,B 0,C 180,E1 -4979.831,E2 -4979.831} C_VEL
LIN {X 0,Y 652.738,Z 286.092,A -85,B 0,C 180,E1 -4982.11,E2 -4982.11} C_VEL
LIN {X 0,Y 654.227,Z 245.943,A -85,B 0,C 180,E1 -4985.076,E2 -4985.076} C_VEL
LIN {X 0,Y 654.341,Z 239.728,A -85,B 0,C 180,E1 -4985.54,E2 -4985.54} C_VEL
LIN {X 0,Y 647.416,Z 221.801,A -85,B 0,C 180,E1 -4987.308,E2 -4987.308} C_VEL
LIN {X 0,Y 640.89,Z 205.935,A -85,B 0,C 180,E1 -4988.8,E2 -4988.8} C_VEL
LIN {X 0,Y 640.804,Z 205.413,A -85,B 0,C 180,E1 -4988.865,E2 -4988.865} C_VEL
LIN {X 0,Y 640.827,Z 205.408,A -85,B 0,C 180,E1 -4991.903,E2 -4991.903} C_VEL
LIN {X 0,Y 640.803,Z 205.411,A -85,B 0,C 180,E1 -4995.021,E2 -4995.021} C_VEL
LIN {X 0,Y 640.822,Z 205.409,A -85,B 0,C 180,E1 -4998.101,E2 -4998.101} C_VEL
LIN {X 0,Y 640.806,Z 205.408,A -85,B 0,C 180,E1 -5001.151,E2 -5001.151} C_VEL
LIN {X 0,Y 640.82,Z 205.406,A -85,B 0,C 180,E1 -5004.23,E2 -5004.23} C_VEL
LIN {X 0,Y 640.81,Z 205.397,A -85,B 0,C 180,E1 -5007.324,E2 -5007.324} C_VEL
LIN {X 0,Y 640.823,Z 205.397,A -85,B 0,C 180,E1 -5010.458,E2 -5010.458} C_VEL
LIN {X 0,Y 640.823,Z 205.406,A -85,B 0,C 180,E1 -5013.596,E2 -5013.596} C_VEL
LIN {X 0,Y 640.826,Z 205.386,A -85,B 0,C 180,E1 -5016.846,E2 -5016.846} C_VEL
LIN {X 0,Y 640.818,Z 205.401,A -85,B 0,C 180,E1 -5020.019,E2 -5020.019} C_VEL
LIN {X 0,Y 640.817,Z 205.393,A -85,B 0,C 180,E1 -5023.129,E2 -5023.129} C_VEL
LIN {X 0,Y 640.81,Z 205.397,A -85,B 0,C 180,E1 -5026.188,E2 -5026.188} C_VEL
LIN {X 0,Y 640.818,Z 205.395,A -85,B 0,C 180,E1 -5029.299,E2 -5029.299} C_VEL
LIN {X 0,Y 640.805,Z 205.398,A -85,B 0,C 180,E1 -5032.378,E2 -5032.378} C_VEL
LIN {X 0,Y 640.819,Z 205.394,A -85,B 0,C 180,E1 -5035.436,E2 -5035.436} C_VEL
LIN {X 0,Y 640.803,Z 205.401,A -85,B 0,C 180,E1 -5038.48,E2 -5038.48} C_VEL
LIN {X 0,Y 640.822,Z 205.388,A -85,B 0,C 180,E1 -5041.52,E2 -5041.52} C_VEL
LIN {X 0,Y 640.801,Z 205.403,A -85,B 0,C 180,E1 -5044.564,E2 -5044.564} C_VEL
LIN {X 0,Y 640.826,Z 205.388,A -85,B 0,C 180,E1 -5047.712,E2 -5047.712} C_VEL
LIN {X 0,Y 640.805,Z 205.403,A -85,B 0,C 180,E1 -5050.792,E2 -5050.792} C_VEL
LIN {X 0,Y 640.82,Z 205.409,A -85,B 0,C 180,E1 -5053.996,E2 -5053.996} C_VEL
LIN {X 0,Y 640.826,Z 205.403,A -85,B 0,C 180,E1 -5057.152,E2 -5057.152} C_VEL
LIN {X 0,Y 640.797,Z 205.408,A -85,B 0,C 180,E1 -5060.316,E2 -5060.316} C_VEL
LIN {X 0,Y 640.834,Z 205.404,A -85,B 0,C 180,E1 -5063.348,E2 -5063.348} C_VEL
LIN {X 0,Y 640.792,Z 205.405,A -85,B 0,C 180,E1 -5066.406,E2 -5066.406} C_VEL
LIN {X 0,Y 640.834,Z 205.402,A -85,B 0,C 180,E1 -5069.466,E2 -5069.466} C_VEL
LIN {X 0,Y 640.786,Z 205.411,A -85,B 0,C 180,E1 -5072.465,E2 -5072.465} C_VEL
LIN {X 0,Y 640.831,Z 205.406,A -85,B 0,C 180,E1 -5075.481,E2 -5075.481} C_VEL
LIN {X 0,Y 640.78,Z 205.411,A -85,B 0,C 180,E1 -5078.577,E2 -5078.577} C_VEL
LIN {X 0,Y 640.835,Z 205.403,A -85,B 0,C 180,E1 -5081.539,E2 -5081.539} C_VEL
LIN {X 0,Y 640.776,Z 205.412,A -85,B 0,C 180,E1 -5084.638,E2 -5084.638} C_VEL
LIN {X 0,Y 642.076,Z 208.877,A -85,B 0,C 180,E1 -5084.992,E2 -5084.992} C_VEL
LIN {X 0,Y 643.369,Z 211.316,A -85,B 0,C 180,E1 -5085.255,E2 -5085.255} C_VEL
LIN {X 0,Y 653.762,Z 232.116,A -85,B 0,C 180,E1 -5087.363,E2 -5087.363} C_VEL
LIN {X 0,Y 660.528,Z 246.496,A -85,B 0,C 180,E1 -5088.704,E2 -5088.704} C_VEL
LIN {X 0,Y 657.722,Z 303.299,A -85,B 0,C 180,E1 -5091.594,E2 -5091.594} C_VEL
LIN {X 0,Y 660.087,Z 320.461,A -85,B 0,C 180,E1 -5091.975,E2 -5091.975} C_VEL
LIN {X 0,Y 657.225,Z 576.361,A -85,B 0,C 180,E1 -5095.111,E2 -5095.111} C_VEL
LIN {X 0,Y 656.033,Z 691.701,A -85,B 0,C 180,E1 -5096.501,E2 -5096.501} C_VEL
LIN {X 0,Y 655.355,Z 717.299,A -85,B 0,C 180,E1 -5096.961,E2 -5096.961} C_VEL
LIN {X 0,Y 654.581,Z 738.856,A -85,B 0,C 180,E1 -5097.482,E2 -5097.482} C_VEL
LIN {X 0,Y 653.482,Z 764.441,A -85,B 0,C 180,E1 -5098.27,E2 -5098.27} C_VEL
LIN {X 0,Y 652.452,Z 785.308,A -85,B 0,C 180,E1 -5099.059,E2 -5099.059} C_VEL
LIN {X 0,Y 651.303,Z 805.277,A -85,B 0,C 180,E1 -5099.968,E2 -5099.968} C_VEL
LIN {X 0,Y 649.76,Z 827.032,A -85,B 0,C 180,E1 -5101.151,E2 -5101.151} C_VEL
LIN {X 0,Y 648.313,Z 847.653,A -85,B 0,C 180,E1 -5102.439,E2 -5102.439} C_VEL
LIN {X 0,Y 646.864,Z 867.215,A -85,B 0,C 180,E1 -5103.862,E2 -5103.862} C_VEL
LIN {X 0,Y 645.559,Z 885.061,A -85,B 0,C 180,E1 -5105.328,E2 -5105.328} C_VEL
LIN {X 0,Y 644.311,Z 902.602,A -85,B 0,C 180,E1 -5106.979,E2 -5106.979} C_VEL
LIN {X 0,Y 643.278,Z 917.865,A -85,B 0,C 180,E1 -5108.602,E2 -5108.602} C_VEL
LIN {X 0,Y 642.3,Z 933.819,A -85,B 0,C 180,E1 -5110.541,E2 -5110.541} C_VEL
LIN {X 0,Y 641.574,Z 946.518,A -85,B 0,C 180,E1 -5112.308,E2 -5112.308} C_VEL
LIN {X 0,Y 640.936,Z 959.769,A -85,B 0,C 180,E1 -5114.435,E2 -5114.435} C_VEL
LIN {X 0,Y 640.537,Z 969.561,A -85,B 0,C 180,E1 -5116.274,E2 -5116.274} C_VEL
LIN {X 0,Y 640.242,Z 979.124,A -85,B 0,C 180,E1 -5118.377,E2 -5118.377} C_VEL
LIN {X 0,Y 640.069,Z 986.514,A -85,B 0,C 180,E1 -5120.378,E2 -5120.378} C_VEL
LIN {X 0,Y 639.945,Z 992.762,A -85,B 0,C 180,E1 -5122.458,E2 -5122.458} C_VEL
LIN {X 0,Y 639.901,Z 997.496,A -85,B 0,C 180,E1 -5124.62,E2 -5124.62} C_VEL
LIN {X 0,Y 639.911,Z 1000.351,A -85,B 0,C 180,E1 -5126.506,E2 -5126.506} C_VEL
LIN {X 0,Y 639.908,Z 1002.192,A -85,B 0,C 180,E1 -5128.747,E2 -5128.747} C_VEL
LIN {X 0,Y 639.885,Z 1002.328,A -85,B 0,C 180,E1 -5130.716,E2 -5130.716} C_VEL
LIN {X 0,Y 639.887,Z 1001.225,A -85,B 0,C 180,E1 -5132.687,E2 -5132.687} C_VEL
LIN {X 0,Y 639.901,Z 998.292,A -85,B 0,C 180,E1 -5134.93,E2 -5134.93} C_VEL
LIN {X 0,Y 639.944,Z 994.689,A -85,B 0,C 180,E1 -5136.73,E2 -5136.73} C_VEL
LIN {X 0,Y 640.007,Z 988.934,A -85,B 0,C 180,E1 -5138.898,E2 -5138.898} C_VEL
LIN {X 0,Y 640.164,Z 981.603,A -85,B 0,C 180,E1 -5140.985,E2 -5140.985} C_VEL
LIN {X 0,Y 640.421,Z 973.53,A -85,B 0,C 180,E1 -5142.901,E2 -5142.901} C_VEL
LIN {X 0,Y 640.82,Z 962.834,A -85,B 0,C 180,E1 -5145.017,E2 -5145.017} C_VEL
LIN {X 0,Y 641.311,Z 951.973,A -85,B 0,C 180,E1 -5146.858,E2 -5146.858} C_VEL
LIN {X 0,Y 642.078,Z 937.321,A -85,B 0,C 180,E1 -5148.994,E2 -5148.994} C_VEL
LIN {X 0,Y 642.89,Z 924.078,A -85,B 0,C 180,E1 -5150.674,E2 -5150.674} C_VEL
LIN {X 0,Y 643.993,Z 907.23,A -85,B 0,C 180,E1 -5152.551,E2 -5152.551} C_VEL
LIN {X 0,Y 645.091,Z 891.542,A -85,B 0,C 180,E1 -5154.083,E2 -5154.083} C_VEL
LIN {X 0,Y 646.455,Z 872.685,A -85,B 0,C 180,E1 -5155.713,E2 -5155.713} C_VEL
LIN {X 0,Y 647.801,Z 854.392,A -85,B 0,C 180,E1 -5157.087,E2 -5157.087} C_VEL
LIN {X 0,Y 649.326,Z 833.594,A -85,B 0,C 180,E1 -5158.463,E2 -5158.463} C_VEL
LIN {X 0,Y 650.699,Z 813.328,A -85,B 0,C 180,E1 -5159.612,E2 -5159.612} C_VEL
LIN {X 0,Y 652.091,Z 792.534,A -85,B 0,C 180,E1 -5160.635,E2 -5160.635} C_VEL
LIN {X 0,Y 653.112,Z 771.457,A -85,B 0,C 180,E1 -5161.471,E2 -5161.471} C_VEL
LIN {X 0,Y 653.982,Z 749.69,A -85,B 0,C 180,E1 -5162.173,E2 -5162.173} C_VEL
LIN {X 0,Y 654.804,Z 724.006,A -85,B 0,C 180,E1 -5162.834,E2 -5162.834} C_VEL
LIN {X 0,Y 655.401,Z 700.977,A -85,B 0,C 180,E1 -5163.275,E2 -5163.275} C_VEL
LIN {X 0,Y 655.819,Z 668.673,A -85,B 0,C 180,E1 -5163.695,E2 -5163.695} C_VEL
LIN {X 0,Y 656.905,Z 438,A -85,B 0,C 180,E1 -5166.286,E2 -5166.286} C_VEL
LIN {X 0,Y 657.494,Z 317.486,A -85,B 0,C 180,E1 -5167.708,E2 -5167.708} C_VEL
LIN {X 0,Y 655.903,Z 308.074,A -85,B 0,C 180,E1 -5167.905,E2 -5167.905} C_VEL
LIN {X 0,Y 657.908,Z 274.941,A -85,B 0,C 180,E1 -5169.667,E2 -5169.667} C_VEL
LIN {X 0,Y 660.829,Z 246.988,A -85,B 0,C 180,E1 -5171.306,E2 -5171.306} C_VEL
LIN {X 0,Y 657.133,Z 237.55,A -85,B 0,C 180,E1 -5172.441,E2 -5172.441} C_VEL
LIN {X 0,Y 653.714,Z 229.544,A -85,B 0,C 180,E1 -5173.657,E2 -5173.657} C_VEL
LIN {X 0,Y 651.418,Z 224.985,A -85,B 0,C 180,E1 -5174.584,E2 -5174.584} C_VEL
LIN {X 0,Y 649.639,Z 221.116,A -85,B 0,C 180,E1 -5175.575,E2 -5175.575} C_VEL
LIN {X 0,Y 647.858,Z 218.188,A -85,B 0,C 180,E1 -5176.888,E2 -5176.888} C_VEL
LIN {X 0,Y 647.588,Z 216.77,A -85,B 0,C 180,E1 -5178.044,E2 -5178.044} C_VEL
LIN {X 0,Y 647.605,Z 217.408,A -85,B 0,C 180,E1 -5179.026,E2 -5179.026} C_VEL
LIN {X 0,Y 648.783,Z 220.148,A -85,B 0,C 180,E1 -5180.407,E2 -5180.407} C_VEL
LIN {X 0,Y 649.676,Z 221.608,A -85,B 0,C 180,E1 -5180.931,E2 -5180.931} C_VEL
LIN {X 0,Y 651.664,Z 226.181,A -85,B 0,C 180,E1 -5182.027,E2 -5182.027} C_VEL
LIN {X 0,Y 654.089,Z 231.929,A -85,B 0,C 180,E1 -5183.082,E2 -5183.082} C_VEL
LIN {X 0,Y 657.229,Z 240.749,A -85,B 0,C 180,E1 -5184.333,E2 -5184.333} C_VEL
LIN {X 0,Y 657.877,Z 243.083,A -85,B 0,C 180,E1 -5184.615,E2 -5184.615} C_VEL
LIN {X 0,Y 654.022,Z 277.586,A -85,B 0,C 180,E1 -5187.07,E2 -5187.07} C_VEL
LIN {X 0,Y 650.667,Z 322.883,A -85,B 0,C 180,E1 -5190.078,E2 -5190.078} C_VEL
LIN {X 0,Y 648.399,Z 368.098,A -85,B 0,C 180,E1 -5192.94,E2 -5192.94} C_VEL
LIN {X 0,Y 646.387,Z 421.369,A -85,B 0,C 180,E1 -5196.188,E2 -5196.188} C_VEL
LIN {X 0,Y 645.642,Z 446.78,A -85,B 0,C 180,E1 -5197.681,E2 -5197.681} C_VEL
LIN {X 0,Y 649.975,Z 484.177,A -85,B 0,C 180,E1 -5198.57,E2 -5198.57} C_VEL
LIN {X 0,Y 646.851,Z 599.918,A -85,B 0,C 180,E1 -5200.294,E2 -5200.294} C_VEL
LIN {X 0,Y 645.385,Z 683.668,A -85,B 0,C 180,E1 -5201.482,E2 -5201.482} C_VEL
LIN {X 0,Y 644.939,Z 704.063,A -85,B 0,C 180,E1 -5201.936,E2 -5201.936} C_VEL
LIN {X 0,Y 644.459,Z 723.235,A -85,B 0,C 180,E1 -5202.529,E2 -5202.529} C_VEL
LIN {X 0,Y 643.922,Z 741.453,A -85,B 0,C 180,E1 -5203.259,E2 -5203.259} C_VEL
LIN {X 0,Y 643.38,Z 759.262,A -85,B 0,C 180,E1 -5204.155,E2 -5204.155} C_VEL
LIN {X 0,Y 642.836,Z 775.536,A -85,B 0,C 180,E1 -5205.161,E2 -5205.161} C_VEL
LIN {X 0,Y 642.318,Z 790.242,A -85,B 0,C 180,E1 -5206.258,E2 -5206.258} C_VEL
LIN {X 0,Y 641.856,Z 803.053,A -85,B 0,C 180,E1 -5207.403,E2 -5207.403} C_VEL
LIN {X 0,Y 641.438,Z 814.956,A -85,B 0,C 180,E1 -5208.673,E2 -5208.673} C_VEL
LIN {X 0,Y 641.059,Z 826.152,A -85,B 0,C 180,E1 -5210.121,E2 -5210.121} C_VEL
LIN {X 0,Y 640.758,Z 835.587,A -85,B 0,C 180,E1 -5211.629,E2 -5211.629} C_VEL
LIN {X 0,Y 640.548,Z 843.291,A -85,B 0,C 180,E1 -5213.187,E2 -5213.187} C_VEL
LIN {X 0,Y 640.415,Z 849.369,A -85,B 0,C 180,E1 -5214.804,E2 -5214.804} C_VEL
LIN {X 0,Y 640.309,Z 853.658,A -85,B 0,C 180,E1 -5216.419,E2 -5216.419} C_VEL
LIN {X 0,Y 640.251,Z 856.386,A -85,B 0,C 180,E1 -5218.121,E2 -5218.121} C_VEL
LIN {X 0,Y 640.222,Z 857.342,A -85,B 0,C 180,E1 -5219.821,E2 -5219.821} C_VEL
LIN {X 0,Y 640.204,Z 856.56,A -85,B 0,C 180,E1 -5221.521,E2 -5221.521} C_VEL
LIN {X 0,Y 640.223,Z 854.029,A -85,B 0,C 180,E1 -5223.223,E2 -5223.223} C_VEL
LIN {X 0,Y 640.273,Z 849.687,A -85,B 0,C 180,E1 -5224.927,E2 -5224.927} C_VEL
LIN {X 0,Y 640.369,Z 843.779,A -85,B 0,C 180,E1 -5226.545,E2 -5226.545} C_VEL
LIN {X 0,Y 640.542,Z 835.96,A -85,B 0,C 180,E1 -5228.167,E2 -5228.167} C_VEL
LIN {X 0,Y 640.802,Z 826.573,A -85,B 0,C 180,E1 -5229.702,E2 -5229.702} C_VEL
LIN {X 0,Y 641.144,Z 815.658,A -85,B 0,C 180,E1 -5231.15,E2 -5231.15} C_VEL
LIN {X 0,Y 641.566,Z 803.212,A -85,B 0,C 180,E1 -5232.511,E2 -5232.511} C_VEL
LIN {X 0,Y 642.071,Z 789.175,A -85,B 0,C 180,E1 -5233.784,E2 -5233.784} C_VEL
LIN {X 0,Y 642.627,Z 773.942,A -85,B 0,C 180,E1 -5234.93,E2 -5234.93} C_VEL
LIN {X 0,Y 643.188,Z 757.942,A -85,B 0,C 180,E1 -5235.925,E2 -5235.925} C_VEL
LIN {X 0,Y 643.745,Z 740.91,A -85,B 0,C 180,E1 -5236.792,E2 -5236.792} C_VEL
LIN {X 0,Y 644.306,Z 722.97,A -85,B 0,C 180,E1 -5237.522,E2 -5237.522} C_VEL
LIN {X 0,Y 644.804,Z 703.329,A -85,B 0,C 180,E1 -5238.132,E2 -5238.132} C_VEL
LIN {X 0,Y 645.21,Z 683.617,A -85,B 0,C 180,E1 -5238.564,E2 -5238.564} C_VEL
LIN {X 0,Y 645.584,Z 652.222,A -85,B 0,C 180,E1 -5238.987,E2 -5238.987} C_VEL
LIN {X 0,Y 647.544,Z 481.946,A -85,B 0,C 180,E1 -5241.13,E2 -5241.13} C_VEL
LIN {X 0,Y 645.194,Z 462.193,A -85,B 0,C 180,E1 -5241.501,E2 -5241.501} C_VEL
LIN {X 0,Y 645.421,Z 453.034,A -85,B 0,C 180,E1 -5242.035,E2 -5242.035} C_VEL
LIN {X 0,Y 644.647,Z 446.758,A -85,B 0,C 180,E1 -5242.435,E2 -5242.435} C_VEL
LIN {X 0,Y 639.241,Z 430.811,A -85,B 0,C 180,E1 -5243.594,E2 -5243.594} C_VEL
LIN {X 0,Y 638.723,Z 425.411,A -85,B 0,C 180,E1 -5243.942,E2 -5243.942} C_VEL
LIN {X 0,Y 640.513,Z 370.69,A -85,B 0,C 180,E1 -5247.219,E2 -5247.219} C_VEL
LIN {X 0,Y 642.235,Z 323.438,A -85,B 0,C 180,E1 -5250.087,E2 -5250.087} C_VEL
LIN {X 0,Y 644.421,Z 269.602,A -85,B 0,C 180,E1 -5253.408,E2 -5253.408} C_VEL
LIN {X 0,Y 645.57,Z 239.683,A -85,B 0,C 180,E1 -5255.291,E2 -5255.291} C_VEL
LIN {X 0,Y 635.215,Z 212.676,A -85,B 0,C 180,E1 -5257.722,E2 -5257.722} C_VEL
LIN {X 0,Y 632.843,Z 206.4,A -85,B 0,C 180,E1 -5258.327,E2 -5258.327} C_VEL
LIN {X 0,Y 632.898,Z 206.394,A -85,B 0,C 180,E1 -5261.372,E2 -5261.372} C_VEL
LIN {X 0,Y 632.88,Z 206.397,A -85,B 0,C 180,E1 -5264.558,E2 -5264.558} C_VEL
LIN {X 0,Y 632.893,Z 206.394,A -85,B 0,C 180,E1 -5267.699,E2 -5267.699} C_VEL
LIN {X 0,Y 632.82,Z 206.401,A -85,B 0,C 180,E1 -5270.683,E2 -5270.683} C_VEL
LIN {X 0,Y 632.849,Z 206.609,A -85,B 0,C 180,E1 -5270.775,E2 -5270.775} C_VEL
LIN {X 0,Y 633.955,Z 209.607,A -85,B 0,C 180,E1 -5271.039,E2 -5271.039} C_VEL
LIN {X 0,Y 641.581,Z 227.74,A -85,B 0,C 180,E1 -5272.793,E2 -5272.793} C_VEL
LIN {X 0,Y 647.552,Z 243.595,A -85,B 0,C 180,E1 -5274.365,E2 -5274.365} C_VEL
LIN {X 0,Y 646.093,Z 282.724,A -85,B 0,C 180,E1 -5277.256,E2 -5277.256} C_VEL
LIN {X 0,Y 645.582,Z 313.879,A -85,B 0,C 180,E1 -5279.422,E2 -5279.422} C_VEL
LIN {X 0,Y 645.792,Z 322.606,A -85,B 0,C 180,E1 -5279.966,E2 -5279.966} C_VEL
LIN {X 0,Y 646.431,Z 327.594,A -85,B 0,C 180,E1 -5280.064,E2 -5280.064} C_VEL
LIN {X 0,Y 644.515,Z 453.18,A -85,B 0,C 180,E1 -5281.649,E2 -5281.649} C_VEL
LIN {X 0,Y 641.737,Z 617.227,A -85,B 0,C 180,E1 -5283.851,E2 -5283.851} C_VEL
LIN {X 0,Y 641.238,Z 639.138,A -85,B 0,C 180,E1 -5284.314,E2 -5284.314} C_VEL
LIN {X 0,Y 640.554,Z 660.587,A -85,B 0,C 180,E1 -5284.925,E2 -5284.925} C_VEL
LIN {X 0,Y 639.803,Z 681.266,A -85,B 0,C 180,E1 -5285.677,E2 -5285.677} C_VEL
LIN {X 0,Y 638.923,Z 701.378,A -85,B 0,C 180,E1 -5286.578,E2 -5286.578} C_VEL
LIN {X 0,Y 637.947,Z 721.125,A -85,B 0,C 180,E1 -5287.656,E2 -5287.656} C_VEL
LIN {X 0,Y 636.947,Z 739.263,A -85,B 0,C 180,E1 -5288.835,E2 -5288.835} C_VEL
LIN {X 0,Y 636.039,Z 755.438,A -85,B 0,C 180,E1 -5290.068,E2 -5290.068} C_VEL
LIN {X 0,Y 635.112,Z 770.997,A -85,B 0,C 180,E1 -5291.457,E2 -5291.457} C_VEL
LIN {X 0,Y 634.324,Z 784.425,A -85,B 0,C 180,E1 -5292.856,E2 -5292.856} C_VEL
LIN {X 0,Y 633.571,Z 798.306,A -85,B 0,C 180,E1 -5294.531,E2 -5294.531} C_VEL
LIN {X 0,Y 632.925,Z 811.14,A -85,B 0,C 180,E1 -5296.385,E2 -5296.385} C_VEL
LIN {X 0,Y 632.559,Z 820.024,A -85,B 0,C 180,E1 -5297.864,E2 -5297.864} C_VEL
LIN {X 0,Y 632.32,Z 827.662,A -85,B 0,C 180,E1 -5299.338,E2 -5299.338} C_VEL
LIN {X 0,Y 632.131,Z 834.521,A -85,B 0,C 180,E1 -5300.899,E2 -5300.899} C_VEL
LIN {X 0,Y 632.009,Z 840.177,A -85,B 0,C 180,E1 -5302.454,E2 -5302.454} C_VEL
LIN {X 0,Y 631.947,Z 844.954,A -85,B 0,C 180,E1 -5304.097,E2 -5304.097} C_VEL
LIN {X 0,Y 631.923,Z 849.065,A -85,B 0,C 180,E1 -5306.008,E2 -5306.008} C_VEL
LIN {X 0,Y 631.916,Z 851.634,A -85,B 0,C 180,E1 -5308.096,E2 -5308.096} C_VEL
LIN {X 0,Y 631.907,Z 852.399,A -85,B 0,C 180,E1 -5309.819,E2 -5309.819} C_VEL
LIN {X 0,Y 631.898,Z 851.988,A -85,B 0,C 180,E1 -5311.451,E2 -5311.451} C_VEL
LIN {X 0,Y 631.903,Z 850.582,A -85,B 0,C 180,E1 -5312.993,E2 -5312.993} C_VEL
LIN {X 0,Y 631.922,Z 847.99,A -85,B 0,C 180,E1 -5314.629,E2 -5314.629} C_VEL
LIN {X 0,Y 631.965,Z 844.23,A -85,B 0,C 180,E1 -5316.267,E2 -5316.267} C_VEL
LIN {X 0,Y 632.015,Z 839.565,A -85,B 0,C 180,E1 -5317.82,E2 -5317.82} C_VEL
LIN {X 0,Y 632.143,Z 833.775,A -85,B 0,C 180,E1 -5319.376,E2 -5319.376} C_VEL
LIN {X 0,Y 632.353,Z 826.338,A -85,B 0,C 180,E1 -5321.03,E2 -5321.03} C_VEL
LIN {X 0,Y 632.74,Z 815.819,A -85,B 0,C 180,E1 -5322.967,E2 -5322.967} C_VEL
LIN {X 0,Y 633.206,Z 804.873,A -85,B 0,C 180,E1 -5324.635,E2 -5324.635} C_VEL
LIN {X 0,Y 633.777,Z 794.037,A -85,B 0,C 180,E1 -5326.095,E2 -5326.095} C_VEL
LIN {X 0,Y 634.431,Z 782.7,A -85,B 0,C 180,E1 -5327.424,E2 -5327.424} C_VEL
LIN {X 0,Y 635.302,Z 767.838,A -85,B 0,C 180,E1 -5328.931,E2 -5328.931} C_VEL
LIN {X 0,Y 636.28,Z 751.126,A -85,B 0,C 180,E1 -5330.37,E2 -5330.37} C_VEL
LIN {X 0,Y 637.196,Z 735.149,A -85,B 0,C 180,E1 -5331.543,E2 -5331.543} C_VEL
LIN {X 0,Y 638.108,Z 717.554,A -85,B 0,C 180,E1 -5332.639,E2 -5332.639} C_VEL
LIN {X 0,Y 639.057,Z 698.199,A -85,B 0,C 180,E1 -5333.661,E2 -5333.661} C_VEL
LIN {X 0,Y 639.905,Z 678.909,A -85,B 0,C 180,E1 -5334.51,E2 -5334.51} C_VEL
LIN {X 0,Y 640.648,Z 658.096,A -85,B 0,C 180,E1 -5335.245,E2 -5335.245} C_VEL
LIN {X 0,Y 641.299,Z 636.268,A -85,B 0,C 180,E1 -5335.845,E2 -5335.845} C_VEL
LIN {X 0,Y 641.783,Z 614.493,A -85,B 0,C 180,E1 -5336.28,E2 -5336.28} C_VEL
LIN {X 0,Y 645.543,Z 392.365,A -85,B 0,C 180,E1 -5339.225,E2 -5339.225} C_VEL
LIN {X 0,Y 646.257,Z 325.008,A -85,B 0,C 180,E1 -5340.069,E2 -5340.069} C_VEL
LIN {X 0,Y 645.682,Z 321.596,A -85,B 0,C 180,E1 -5340.166,E2 -5340.166} C_VEL
LIN {X 0,Y 645.872,Z 291.858,A -85,B 0,C 180,E1 -5342.178,E2 -5342.178} C_VEL
LIN {X 0,Y 647.35,Z 249.543,A -85,B 0,C 180,E1 -5345.287,E2 -5345.287} C_VEL
LIN {X 0,Y 647.501,Z 243.241,A -85,B 0,C 180,E1 -5345.757,E2 -5345.757} C_VEL
LIN {X 0,Y 640.016,Z 223.753,A -85,B 0,C 180,E1 -5347.692,E2 -5347.692} C_VEL
LIN {X 0,Y 633.801,Z 209.288,A -85,B 0,C 180,E1 -5349.087,E2 -5349.087} C_VEL
LIN {X 0,Y 632.869,Z 206.401,A -85,B 0,C 180,E1 -5349.356,E2 -5349.356} C_VEL
LIN {X 0,Y 632.883,Z 206.396,A -85,B 0,C 180,E1 -5352.588,E2 -5352.588} C_VEL
LIN {X 0,Y 632.889,Z 206.394,A -85,B 0,C 180,E1 -5355.708,E2 -5355.708} C_VEL
LIN {X 0,Y 632.87,Z 206.396,A -85,B 0,C 180,E1 -5358.909,E2 -5358.909} C_VEL
LIN {X 0,Y 632.884,Z 206.393,A -85,B 0,C 180,E1 -5361.964,E2 -5361.964} C_VEL
LIN {X 0,Y 632.87,Z 206.395,A -85,B 0,C 180,E1 -5365.115,E2 -5365.115} C_VEL
LIN {X 0,Y 632.88,Z 206.394,A -85,B 0,C 180,E1 -5368.21,E2 -5368.21} C_VEL
LIN {X 0,Y 632.872,Z 206.386,A -85,B 0,C 180,E1 -5371.266,E2 -5371.266} C_VEL
LIN {X 0,Y 632.879,Z 206.391,A -85,B 0,C 180,E1 -5374.348,E2 -5374.348} C_VEL
LIN {X 0,Y 632.88,Z 206.382,A -85,B 0,C 180,E1 -5377.521,E2 -5377.521} C_VEL
LIN {X 0,Y 632.888,Z 206.382,A -85,B 0,C 180,E1 -5380.719,E2 -5380.719} C_VEL
LIN {X 0,Y 632.883,Z 206.396,A -85,B 0,C 180,E1 -5383.95,E2 -5383.95} C_VEL
LIN {X 0,Y 632.882,Z 206.381,A -85,B 0,C 180,E1 -5387.11,E2 -5387.11} C_VEL
LIN {X 0,Y 632.871,Z 206.396,A -85,B 0,C 180,E1 -5390.175,E2 -5390.175} C_VEL
LIN {X 0,Y 632.881,Z 206.384,A -85,B 0,C 180,E1 -5393.286,E2 -5393.286} C_VEL
LIN {X 0,Y 632.866,Z 206.395,A -85,B 0,C 180,E1 -5396.377,E2 -5396.377} C_VEL
LIN {X 0,Y 632.882,Z 206.387,A -85,B 0,C 180,E1 -5399.457,E2 -5399.457} C_VEL
LIN {X 0,Y 632.863,Z 206.392,A -85,B 0,C 180,E1 -5402.536,E2 -5402.536} C_VEL
LIN {X 0,Y 632.888,Z 206.386,A -85,B 0,C 180,E1 -5405.712,E2 -5405.712} C_VEL
LIN {X 0,Y 632.869,Z 206.387,A -85,B 0,C 180,E1 -5408.816,E2 -5408.816} C_VEL
LIN {X 0,Y 632.875,Z 206.399,A -85,B 0,C 180,E1 -5412.049,E2 -5412.049} C_VEL
LIN {X 0,Y 632.895,Z 206.388,A -85,B 0,C 180,E1 -5415.204,E2 -5415.204} C_VEL
LIN {X 0,Y 632.858,Z 206.394,A -85,B 0,C 180,E1 -5418.325,E2 -5418.325} C_VEL
LIN {X 0,Y 632.894,Z 206.391,A -85,B 0,C 180,E1 -5421.405,E2 -5421.405} C_VEL
LIN {X 0,Y 632.851,Z 206.397,A -85,B 0,C 180,E1 -5424.485,E2 -5424.485} C_VEL
LIN {X 0,Y 632.893,Z 206.391,A -85,B 0,C 180,E1 -5427.587,E2 -5427.587} C_VEL
LIN {X 0,Y 632.847,Z 206.398,A -85,B 0,C 180,E1 -5430.581,E2 -5430.581} C_VEL
LIN {X 0,Y 632.894,Z 206.393,A -85,B 0,C 180,E1 -5433.679,E2 -5433.679} C_VEL
LIN {X 0,Y 632.842,Z 206.399,A -85,B 0,C 180,E1 -5436.673,E2 -5436.673} C_VEL
LIN {X 0,Y 632.896,Z 206.392,A -85,B 0,C 180,E1 -5439.7,E2 -5439.7} C_VEL
LIN {X 0,Y 632.838,Z 206.402,A -85,B 0,C 180,E1 -5442.718,E2 -5442.718} C_VEL
LIN {X 0,Y 632.9,Z 206.535,A -85,B 0,C 180,E1 -5444.042,E2 -5444.042} C_VEL
LIN {X 0,Y 633.936,Z 209.536,A -85,B 0,C 180,E1 -5444.326,E2 -5444.326} C_VEL
LIN {X 0,Y 635.232,Z 211.906,A -85,B 0,C 180,E1 -5444.59,E2 -5444.59} C_VEL
LIN {X 0,Y 645.759,Z 232.745,A -85,B 0,C 180,E1 -5446.763,E2 -5446.763} C_VEL
LIN {X 0,Y 653.974,Z 250.328,A -85,B 0,C 180,E1 -5448.428,E2 -5448.428} C_VEL
LIN {X 0,Y 651.046,Z 303.925,A -85,B 0,C 180,E1 -5451.191,E2 -5451.191} C_VEL
LIN {X 0,Y 653.477,Z 321.86,A -85,B 0,C 180,E1 -5451.594,E2 -5451.594} C_VEL
LIN {X 0,Y 650.878,Z 527.556,A -85,B 0,C 180,E1 -5454.159,E2 -5454.159} C_VEL
LIN {X 0,Y 648.936,Z 692.545,A -85,B 0,C 180,E1 -5456.184,E2 -5456.184} C_VEL
LIN {X 0,Y 648.205,Z 717.768,A -85,B 0,C 180,E1 -5456.648,E2 -5456.648} C_VEL
LIN {X 0,Y 647.368,Z 739.572,A -85,B 0,C 180,E1 -5457.184,E2 -5457.184} C_VEL
LIN {X 0,Y 646.169,Z 765.275,A -85,B 0,C 180,E1 -5457.993,E2 -5457.993} C_VEL
LIN {X 0,Y 645.045,Z 786.711,A -85,B 0,C 180,E1 -5458.819,E2 -5458.819} C_VEL
LIN {X 0,Y 643.662,Z 810.452,A -85,B 0,C 180,E1 -5459.914,E2 -5459.914} C_VEL
LIN {X 0,Y 642.593,Z 827.04,A -85,B 0,C 180,E1 -5460.801,E2 -5460.801} C_VEL
LIN {X 0,Y 641.236,Z 844.718,A -85,B 0,C 180,E1 -5461.906,E2 -5461.906} C_VEL
LIN {X 0,Y 639.571,Z 865.996,A -85,B 0,C 180,E1 -5463.441,E2 -5463.441} C_VEL
LIN {X 0,Y 638.241,Z 882.84,A -85,B 0,C 180,E1 -5464.828,E2 -5464.828} C_VEL
LIN {X 0,Y 636.789,Z 901.674,A -85,B 0,C 180,E1 -5466.593,E2 -5466.593} C_VEL
LIN {X 0,Y 635.682,Z 916.781,A -85,B 0,C 180,E1 -5468.21,E2 -5468.21} C_VEL
LIN {X 0,Y 634.573,Z 933.116,A -85,B 0,C 180,E1 -5470.198,E2 -5470.198} C_VEL
LIN {X 0,Y 633.767,Z 945.881,A -85,B 0,C 180,E1 -5471.987,E2 -5471.987} C_VEL
LIN {X 0,Y 633.093,Z 958.731,A -85,B 0,C 180,E1 -5474.049,E2 -5474.049} C_VEL
LIN {X 0,Y 632.626,Z 969.101,A -85,B 0,C 180,E1 -5476.006,E2 -5476.006} C_VEL
LIN {X 0,Y 632.302,Z 978.77,A -85,B 0,C 180,E1 -5478.137,E2 -5478.137} C_VEL
LIN {X 0,Y 632.087,Z 986.211,A -85,B 0,C 180,E1 -5480.163,E2 -5480.163} C_VEL
LIN {X 0,Y 631.97,Z 991.999,A -85,B 0,C 180,E1 -5482.088,E2 -5482.088} C_VEL
LIN {X 0,Y 631.917,Z 997.176,A -85,B 0,C 180,E1 -5484.37,E2 -5484.37} C_VEL
LIN {X 0,Y 631.915,Z 1000.124,A -85,B 0,C 180,E1 -5486.28,E2 -5486.28} C_VEL
LIN {X 0,Y 631.899,Z 1002.103,A -85,B 0,C 180,E1 -5488.459,E2 -5488.459} C_VEL
LIN {X 0,Y 631.884,Z 1002.373,A -85,B 0,C 180,E1 -5490.544,E2 -5490.544} C_VEL
LIN {X 0,Y 631.901,Z 1001.428,A -85,B 0,C 180,E1 -5492.449,E2 -5492.449} C_VEL
LIN {X 0,Y 631.914,Z 998.768,A -85,B 0,C 180,E1 -5494.72,E2 -5494.72} C_VEL
LIN {X 0,Y 631.945,Z 994.895,A -85,B 0,C 180,E1 -5496.724,E2 -5496.724} C_VEL
LIN {X 0,Y 632.003,Z 989.71,A -85,B 0,C 180,E1 -5498.736,E2 -5498.736} C_VEL
LIN {X 0,Y 632.177,Z 982.308,A -85,B 0,C 180,E1 -5500.941,E2 -5500.941} C_VEL
LIN {X 0,Y 632.428,Z 974.751,A -85,B 0,C 180,E1 -5502.788,E2 -5502.788} C_VEL
LIN {X 0,Y 632.849,Z 964.405,A -85,B 0,C 180,E1 -5504.924,E2 -5504.924} C_VEL
LIN {X 0,Y 633.384,Z 953.117,A -85,B 0,C 180,E1 -5506.886,E2 -5506.886} C_VEL
LIN {X 0,Y 634.153,Z 939.764,A -85,B 0,C 180,E1 -5508.907,E2 -5508.907} C_VEL
LIN {X 0,Y 635.062,Z 925.617,A -85,B 0,C 180,E1 -5510.748,E2 -5510.748} C_VEL
LIN {X 0,Y 636.186,Z 909.998,A -85,B 0,C 180,E1 -5512.55,E2 -5512.55} C_VEL
LIN {X 0,Y 637.46,Z 892.822,A -85,B 0,C 180,E1 -5514.265,E2 -5514.265} C_VEL
LIN {X 0,Y 638.907,Z 874.495,A -85,B 0,C 180,E1 -5515.889,E2 -5515.889} C_VEL
LIN {X 0,Y 640.439,Z 855.057,A -85,B 0,C 180,E1 -5517.374,E2 -5517.374} C_VEL
LIN {X 0,Y 642.047,Z 834.746,A -85,B 0,C 180,E1 -5518.742,E2 -5518.742} C_VEL
LIN {X 0,Y 643.264,Z 816.477,A -85,B 0,C 180,E1 -5519.777,E2 -5519.777} C_VEL
LIN {X 0,Y 644.351,Z 796.553,A -85,B 0,C 180,E1 -5520.718,E2 -5520.718} C_VEL
LIN {X 0,Y 645.536,Z 772.741,A -85,B 0,C 180,E1 -5521.674,E2 -5521.674} C_VEL
LIN {X 0,Y 646.466,Z 750.59,A -85,B 0,C 180,E1 -5522.402,E2 -5522.402} C_VEL
LIN {X 0,Y 647.321,Z 725.958,A -85,B 0,C 180,E1 -5523.056,E2 -5523.056} C_VEL
LIN {X 0,Y 647.966,Z 701.892,A -85,B 0,C 180,E1 -5523.528,E2 -5523.528} C_VEL
LIN {X 0,Y 648.405,Z 672.909,A -85,B 0,C 180,E1 -5523.919,E2 -5523.919} C_VEL
LIN {X 0,Y 649.549,Z 453.207,A -85,B 0,C 180,E1 -5526.408,E2 -5526.408} C_VEL
LIN {X 0,Y 650.483,Z 318.941,A -85,B 0,C 180,E1 -5528.025,E2 -5528.025} C_VEL
LIN {X 0,Y 649.032,Z 309.647,A -85,B 0,C 180,E1 -5528.238,E2 -5528.238} C_VEL
LIN {X 0,Y 651.379,Z 277.525,A -85,B 0,C 180,E1 -5530.005,E2 -5530.005} C_VEL
LIN {X 0,Y 654.506,Z 251.306,A -85,B 0,C 180,E1 -5531.589,E2 -5531.589} C_VEL
LIN {X 0,Y 652.582,Z 245.471,A -85,B 0,C 180,E1 -5532.271,E2 -5532.271} C_VEL
LIN {X 0,Y 649.431,Z 237.865,A -85,B 0,C 180,E1 -5533.388,E2 -5533.388} C_VEL
LIN {X 0,Y 646.808,Z 231.657,A -85,B 0,C 180,E1 -5534.549,E2 -5534.549} C_VEL
LIN {X 0,Y 644.659,Z 227.282,A -85,B 0,C 180,E1 -5535.736,E2 -5535.736} C_VEL
LIN {X 0,Y 643.167,Z 224.433,A -85,B 0,C 180,E1 -5537.083,E2 -5537.083} C_VEL
LIN {X 0,Y 643.014,Z 223.304,A -85,B 0,C 180,E1 -5538.156,E2 -5538.156} C_VEL
LIN {X 0,Y 642.996,Z 224.118,A -85,B 0,C 180,E1 -5539.105,E2 -5539.105} C_VEL
LIN {X 0,Y 644.221,Z 226.82,A -85,B 0,C 180,E1 -5540.479,E2 -5540.479} C_VEL
LIN {X 0,Y 644.754,Z 227.969,A -85,B 0,C 180,E1 -5540.863,E2 -5540.863} C_VEL
LIN {X 0,Y 646.517,Z 232.246,A -85,B 0,C 180,E1 -5541.926,E2 -5541.926} C_VEL
LIN {X 0,Y 648.723,Z 237.823,A -85,B 0,C 180,E1 -5542.978,E2 -5542.978} C_VEL
LIN {X 0,Y 651.64,Z 246.685,A -85,B 0,C 180,E1 -5544.263,E2 -5544.263} C_VEL
LIN {X 0,Y 648.257,Z 273.291,A -85,B 0,C 180,E1 -5546.24,E2 -5546.24} C_VEL
LIN {X 0,Y 644.469,Z 314.816,A -85,B 0,C 180,E1 -5549.1,E2 -5549.1} C_VEL
LIN {X 0,Y 641.686,Z 361.357,A -85,B 0,C 180,E1 -5552.13,E2 -5552.13} C_VEL
LIN {X 0,Y 639.385,Z 412.532,A -85,B 0,C 180,E1 -5555.32,E2 -5555.32} C_VEL
LIN {X 0,Y 638.327,Z 443.948,A -85,B 0,C 180,E1 -5557.204,E2 -5557.204} C_VEL
LIN {X 0,Y 642.421,Z 479.638,A -85,B 0,C 180,E1 -5558.104,E2 -5558.104} C_VEL
LIN {X 0,Y 642.916,Z 487.294,A -85,B 0,C 180,E1 -5558.266,E2 -5558.266} C_VEL
LIN {X 0,Y 639.482,Z 602.556,A -85,B 0,C 180,E1 -5560.041,E2 -5560.041} C_VEL
LIN {X 0,Y 637.883,Z 684.332,A -85,B 0,C 180,E1 -5561.24,E2 -5561.24} C_VEL
LIN {X 0,Y 637.375,Z 705.209,A -85,B 0,C 180,E1 -5561.72,E2 -5561.72} C_VEL
LIN {X 0,Y 636.827,Z 725.235,A -85,B 0,C 180,E1 -5562.36,E2 -5562.36} C_VEL
LIN {X 0,Y 636.236,Z 743.839,A -85,B 0,C 180,E1 -5563.13,E2 -5563.13} C_VEL
LIN {X 0,Y 635.678,Z 761.117,A -85,B 0,C 180,E1 -5564.022,E2 -5564.022} C_VEL
LIN {X 0,Y 635.104,Z 777.203,A -85,B 0,C 180,E1 -5565.037,E2 -5565.037} C_VEL
LIN {X 0,Y 634.553,Z 791.727,A -85,B 0,C 180,E1 -5566.142,E2 -5566.142} C_VEL
LIN {X 0,Y 634.047,Z 804.854,A -85,B 0,C 180,E1 -5567.338,E2 -5567.338} C_VEL
LIN {X 0,Y 633.605,Z 816.656,A -85,B 0,C 180,E1 -5568.623,E2 -5568.623} C_VEL
LIN {X 0,Y 633.221,Z 827.13,A -85,B 0,C 180,E1 -5569.997,E2 -5569.997} C_VEL
LIN {X 0,Y 632.901,Z 836.416,A -85,B 0,C 180,E1 -5571.49,E2 -5571.49} C_VEL
LIN {X 0,Y 632.672,Z 843.948,A -85,B 0,C 180,E1 -5573.01,E2 -5573.01} C_VEL
LIN {X 0,Y 632.518,Z 850.147,A -85,B 0,C 180,E1 -5574.648,E2 -5574.648} C_VEL
LIN {X 0,Y 632.398,Z 854.536,A -85,B 0,C 180,E1 -5576.283,E2 -5576.283} C_VEL
LIN {X 0,Y 632.326,Z 857.346,A -85,B 0,C 180,E1 -5578.006,E2 -5578.006} C_VEL
LIN {X 0,Y 632.291,Z 858.371,A -85,B 0,C 180,E1 -5579.728,E2 -5579.728} C_VEL
LIN {X 0,Y 632.271,Z 857.643,A -85,B 0,C 180,E1 -5581.45,E2 -5581.45} C_VEL
LIN {X 0,Y 632.288,Z 855.157,A -85,B 0,C 180,E1 -5583.173,E2 -5583.173} C_VEL
LIN {X 0,Y 632.334,Z 851.122,A -85,B 0,C 180,E1 -5584.807,E2 -5584.807} C_VEL
LIN {X 0,Y 632.435,Z 845.351,A -85,B 0,C 180,E1 -5586.445,E2 -5586.445} C_VEL
LIN {X 0,Y 632.606,Z 837.68,A -85,B 0,C 180,E1 -5588.087,E2 -5588.087} C_VEL
LIN {X 0,Y 632.877,Z 828.445,A -85,B 0,C 180,E1 -5589.644,E2 -5589.644} C_VEL
LIN {X 0,Y 633.234,Z 817.757,A -85,B 0,C 180,E1 -5591.107,E2 -5591.107} C_VEL
LIN {X 0,Y 633.675,Z 805.564,A -85,B 0,C 180,E1 -5592.485,E2 -5592.485} C_VEL
LIN {X 0,Y 634.214,Z 791.659,A -85,B 0,C 180,E1 -5593.79,E2 -5593.79} C_VEL
LIN {X 0,Y 634.805,Z 776.472,A -85,B 0,C 180,E1 -5594.97,E2 -5594.97} C_VEL
LIN {X 0,Y 635.425,Z 759.895,A -85,B 0,C 180,E1 -5596.031,E2 -5596.031} C_VEL
LIN {X 0,Y 636.005,Z 743.177,A -85,B 0,C 180,E1 -5596.909,E2 -5596.909} C_VEL
LIN {X 0,Y 636.595,Z 725.725,A -85,B 0,C 180,E1 -5597.647,E2 -5597.647} C_VEL
LIN {X 0,Y 637.118,Z 706.586,A -85,B 0,C 180,E1 -5598.273,E2 -5598.273} C_VEL
LIN {X 0,Y 637.572,Z 687.079,A -85,B 0,C 180,E1 -5598.733,E2 -5598.733} C_VEL
LIN {X 0,Y 637.92,Z 664.257,A -85,B 0,C 180,E1 -5599.076,E2 -5599.076} C_VEL
LIN {X 0,Y 640.189,Z 482.959,A -85,B 0,C 180,E1 -5601.398,E2 -5601.398} C_VEL
LIN {X 0,Y 637.648,Z 461.325,A -85,B 0,C 180,E1 -5601.817,E2 -5601.817} C_VEL
LIN {X 0,Y 638.723,Z 425.411,A -85,B 0,C 180,E1 -5603.942,E2 -5603.942} C_VEL
LIN {X 0,Y 638.011,Z 419.163,A -85,B 0,C 180,E1 -5604.35,E2 -5604.35} C_VEL
LIN {X 0,Y 632.689,Z 403.351,A -85,B 0,C 180,E1 -5605.54,E2 -5605.54} C_VEL
LIN {X 0,Y 632.169,Z 397.972,A -85,B 0,C 180,E1 -5605.894,E2 -5605.894} C_VEL
LIN {X 0,Y 634.213,Z 344.412,A -85,B 0,C 180,E1 -5609.155,E2 -5609.155} C_VEL
